  // ------------------------------------------
  // Write data from PLC to RC
  // ------------------------------------------
  30 : IF (( NOT _writeRobotReferenceDynamics.Busy  ) AND 
           ( NOT _writeRobotReferenceDynamics.Error ))
       THEN
         // set command parameter
        _writeRobotReferenceDynamics.ParCmd.DynamicValues :=  ReferenceDynamics;
         // execute command
        _writeRobotReferenceDynamics.Execute := TRUE;
         // set timeout
         SetTimeout(PT := _rTimeout, rTimer := _rTimer);
         // inc step counter
        _rStep := _rStep + 1;
       ELSE
         // check error ? 
         IF (_writeRobotReferenceDynamics.Error)
         THEN
           ErrorID     := _writeRobotReferenceDynamics.ErrorID;
           ErrorAddTxt := _writeRobotReferenceDynamics.ErrorAddTxt;;
         END_IF  
       
         // timeout exceeded ? 
         IF (CheckTimeout(_rTimer) = RobotLibraryConstants.OK)
         THEN
           ErrorID     := RobotLibraryErrorIdEnum.ERR_TIMEOUT_CMD;
           ErrorAddTxt := CONCAT(_stepName, DINT_TO_STRING(_rStep));
         END_IF
       END_IF
 
  31 : IF (( NOT _writeRobotReferenceDynamics.Busy  ) AND
           ( NOT _writeRobotReferenceDynamics.Error ) AND
           (     _writeRobotReferenceDynamics.Done  ))
       THEN
         // execute command
        _writeRobotReferenceDynamics.Execute := FALSE;      
         // update internal ReferenceDynamics data
        _ReferenceDynamics := ReferenceDynamics; 
         // set timeout
         SetTimeout(PT := _rTimeout, rTimer := _rTimer);
         // inc step counter
        _rStep := 10; // -> jump to after startup;           
       ELSE
         // check error ? 
         IF (_writeRobotReferenceDynamics.Error)
         THEN
           SetWarning( WarningID := RobotLibraryWarningIdEnum.WARN_REFERENCE_DYNAMICS_SYNC_FAILED_BY_ERROR_OF_READ_OR_WRITE_CMD, Overwrite := TRUE);    
         END_IF  
       
         // timeout exceeded ? 
         IF (CheckTimeout(_rTimer) = RobotLibraryConstants.OK)
         THEN
           ErrorID     := RobotLibraryErrorIdEnum.ERR_TIMEOUT_CMD;
           ErrorAddTxt := CONCAT(_stepName, DINT_TO_STRING(_rStep));
         END_IF
       END_IF
       
ELSE
  // invalid step
  ErrorID     := RobotLibraryErrorIdEnum.ERR_INVALID_STEP;
  ErrorAddTxt := CONCAT(_stepName , DINT_TO_STRING(_stepCmd));
END_CASE  
                
END_METHOD

METHOD PRIVATE HandleSyncRobotSWLimits
VAR_IN_OUT
   /// Robot assignment of function
  AxesGroup : AxesGroup;
  /// Software limits stored on PLC
  SWLimits  : SWLimits;
END_VAR 

VAR
  /// Internal step counter name
 _stepName        : STRING;    
  /// Internal reference to step counter
 _rStep           : REFERENCE TO DINT;
  /// Internal reference to timer
 _rTimer          : REFERENCE TO TON;
  /// Internal reference to timeout
 _rTimeout        : REFERENCE TO TIME; 
  /// empty data set to reset all DataChanged bits
 _dataChangedNone : AxesGroupStateDataChanged;
END_VAR
                  // Set internal references 
_stepName      :=   '_stepSyncSWLimits = ';
_rStep       REF=    _stepSyncSWLimits;
_rTimer      REF=   _timerSyncSWLimits;
_rTimeout    REF= _timeoutSyncSWLimits;

CASE _rStep
OF    
  0: // Check initialisation configured ?
     IF (( _parCfg.PLC.Parameter.SynchronizationModes.SWLimits[SyncTime.DURING_START_UP] = SyncMode.NO_SYNCHRONIZATION ) AND
         ( _parCfg.PLC.Parameter.SynchronizationModes.SWLimits[SyncTime. AFTER_START_UP] = SyncMode.NO_SYNCHRONIZATION ))
     THEN
       RETURN;
     END_IF

     // Check RC function for sync mode is available ?  
     IF  ((  AxesGroup.State.Initialized                                                  = TRUE                      ) AND  
          (  AxesGroup.State.RobotData.RCSupportedFunctions.WriteRobotSWLimits            = FALSE                     ) AND
         (( _parCfg.PLC.Parameter.SynchronizationModes.SWLimits[SyncTime.DURING_START_UP] = SyncMode.CLIENT_TO_SERVER ) OR
          ( _parCfg.PLC.Parameter.SynchronizationModes.SWLimits[SyncTime. AFTER_START_UP] = SyncMode.CLIENT_TO_SERVER ) OR
          ( _parCfg.PLC.Parameter.SynchronizationModes.SWLimits[SyncTime. AFTER_START_UP] = SyncMode.AUTOMATIC        )))
     THEN
       SetError( ErrorID := RobotLibraryErrorIdEnum.ERR_SYNC_MODE_INVALID, Overwrite := FALSE);
       // Create log entry
       CreateLogMessagePara1 ( Timestamp   := SystemTime,
                               MessageType := MessageType.CMD,
                               Severity    := Severity.DEBUG,
                               MessageCode := 0,
                               MessageText := 'HandleSyncRobotSWLimits: SyncMode needs WriteRobotSWLimits function which is not available on RC',
                               Para1       :=  '');
       RETURN;
     END_IF

     // wait for initialisation done
     IF  ((     AxesGroup.State.RobotData.RCSupportedFunctions .ReadRobotSWLimits ) AND //  ReadRobotSwLimits is mandatory
     //   (     AxesGroup.State.RobotData.RCSupportedFunctions.WriteRobotSWLimits ) AND // WriteRobotSwLimits is optional
          (     AxesGroup.State.Initialized                                       ) AND 
          ( NOT Error                                                             ))  
     THEN
       // Create log entry
       CreateLogMessagePara1 ( Timestamp   := SystemTime,
                               MessageType := MessageType.CMD,
                               Severity    := Severity.DEBUG,
                               MessageCode := 0,
                               MessageText := 'SyncSwLimits: Start initial reading of SwLimits from RC',
                               Para1       :=  '');
       
       // set timeout
       SetTimeout(PT := _rTimeout, rTimer := _rTimer);
       // inc step counter
      _rStep := _rStep + 1;
     END_IF     

     
     // Start read SwLimits
  1: IF (( NOT _readRobotSWLimits.Busy  ) AND 
         ( NOT _readRobotSWLimits.Error ) AND
         ( NOT _readRobotSWLimits.Done  ))
     THEN
       // execute command
      _readRobotSWLimits.Execute := TRUE;
       // set timeout
       SetTimeout(PT := _rTimeout, rTimer := _rTimer);
       // inc step counter
      _rStep := _rStep + 1;
     ELSE
       // check error ? 
       IF ( _readRobotSWLimits.Error )
       THEN
         SetWarning ( WarningID := RobotLibraryWarningIdEnum.WARN_SW_LIMITS_SYNC_FAILED_BY_ERROR_OF_READ_OR_WRITE_CMD, Overwrite := FALSE );           
       END_IF  
       
       // timeout exceeded ? 
       IF (CheckTimeout(_rTimer) = RobotLibraryConstants.OK)
       THEN
         ErrorID     := RobotLibraryErrorIdEnum.ERR_TIMEOUT_CMD;
         ErrorAddTxt := CONCAT(_stepName, DINT_TO_STRING(_rStep));
       END_IF
     END_IF
 
     
     // Wait SwLimits read
  2: IF (( NOT _readRobotSWLimits.Busy  ) AND
         ( NOT _readRobotSWLimits.Error ) AND
         (     _readRobotSWLimits.Done  ))
     THEN
       // reset execution
      _readRobotSWLimits.Execute := FALSE;
       // Copy data
      _swLimits := _readRobotSWLimits.OutCmd.LimitValues;
       // Set plc in sync flag
       AxesGroup.State.SyncStatePlc.InSync.SwLimits := TRUE;
       // inc step counter
      _rStep := _rStep + 1;           

       // Check SwLimits data is equal ? 
       IF ( NOT IsSwLimitsEqual( Data1 := _swLimits, Data2 := SwLimits, IgnoreTimestamp := TRUE))
       THEN
         // Reset plc in sync flag
         AxesGroup.State.SyncStatePlc.InSync.SwLimits := FALSE;
         // Set data changed flag
         AxesGroup.State.DataChanged.SwLimits := TRUE;
         // set timeout
         SetTimeout(PT := _rTimeout, rTimer := _rTimer);
        
         // Create log entry
         CreateLogMessagePara1 ( Timestamp   := SystemTime,
                                 MessageType := MessageType.CMD,
                                 Severity    := Severity.DEBUG,
                                 MessageCode := 0,
                                 MessageText := 'SyncSwLimits: Detected a difference in SwLimits between PLC and RC',
                                 Para1       :=  '');
        
        
         // Check synchronisation is enabled ? 
         IF ( NOT  AxesGroup.State.DataEnableSync.EnableSyncSWLimits )
         THEN
           SetInfo( InfoID := RobotLibraryInfoIdEnum.INFO_SYNC_SWLIMIT_DISABLED, Overwrite := FALSE );
				 END_IF
         
         // Check user interaction needed ?  
         IF ( AxesGroup.Parameter.Plc.Parameter.SyncUserInteraction.SWLimits )
         THEN
           SetWarning ( WarningID := RobotLibraryWarningIdEnum.WARN_SW_LIMITS_SYNC_ERROR, Overwrite := FALSE );                    
				 END_IF
			 END_IF             
     ELSE
       // check error ? 
       IF (_readRobotSWLimits.Error)
       THEN
         // Set warning
         SetWarning( WarningID := RobotLibraryWarningIdEnum.WARN_SW_LIMITS_SYNC_FAILED_BY_ERROR_OF_READ_OR_WRITE_CMD, Overwrite := TRUE);                    
       END_IF  
       
       // timeout exceeded ? 
       IF (CheckTimeout(_rTimer) = RobotLibraryConstants.OK)
       THEN
         ErrorID     := RobotLibraryErrorIdEnum.ERR_TIMEOUT_CMD;
         ErrorAddTxt := CONCAT(_stepName, DINT_TO_STRING(_rStep));
       END_IF
     END_IF
     
     
     // Check synchronisation state ? 
  3: IF ((  NOT AxesGroup.State.DataChanged.SwLimits                                                                                    ) OR 
         (      AxesGroup.Parameter.Plc.Parameter.SynchronizationModes.SWLimits[SyncTime.DURING_START_UP] = SyncMode.NO_SYNCHRONIZATION ))
     THEN
       // Update bit for data in sync
       AxesGroup.State.SyncStatePlc.InSync.SwLimits := NOT AxesGroup.State.DataChanged.SwLimits ;
       // set timeout
       SetTimeout(PT := _rTimeout, rTimer := _rTimer);
       // inc step counter
      _rStep := 10; // -> jump to after startup
            
       // Create log entry
       CreateLogMessagePara1 ( Timestamp   := SystemTime,
                               MessageType := MessageType.CMD,
                               Severity    := Severity.DEBUG,
                               MessageCode := 0,
                               MessageText := 'SyncSwLimits: Synchronization Startup Phase done',
                               Para1       :=  '' );      
     ELSE 
       // Check user interaction needed ? 
       IF ( NOT AxesGroup.Parameter.Plc.Parameter.SyncUserInteraction.SWLimits )
       THEN 
         CASE AxesGroup.Parameter.Plc.Parameter.SynchronizationModes.SWLimits[SyncTime.DURING_START_UP] OF

           SyncMode.SERVER_TO_CLIENT : 

             // Overwrite PLC data with RC data
             SwLimits := _swLimits;            
             // Reset data changed flags
             AxesGroup.State.DataChanged.SwLimits := _dataChangedNone.SwLimits;
             // Reset Synchronizing flag
             AxesGroup.State.Synchronizing.SwLimits := FALSE;
             // Set plc in sync flag
             AxesGroup.State.SyncStatePlc.InSync.SwLimits := TRUE;
             // set timeout
             SetTimeout(PT := _rTimeout, rTimer := _rTimer);
             // inc step counter
            _rStep := 10; // -> jump to after startup         

            // Create log entry
            CreateLogMessagePara2 ( Timestamp   := SystemTime,
                                    MessageType := MessageType.CMD,
                                    Severity    := Severity.DEBUG,
                                    MessageCode := 0,
                                    MessageText := 'SyncSwLimits: Synchronization of SwLimits triggered by StartUp-Compare, SyncMode = {1}, SyncTime = {2}, SyncDirection = RC -> PLC',
                                    Para1       :=  SYNC_MODE_TO_STRING(AxesGroup.Parameter.Plc.Parameter.SynchronizationModes.SWLimits[SyncTime.DURING_START_UP]),
                                    Para2       :=  SYNC_TIME_TO_STRING(SyncTime.DURING_START_UP));
            // Create log entry
            CreateLogMessagePara1 ( Timestamp   := SystemTime,
                                    MessageType := MessageType.CMD,
                                    Severity    := Severity.DEBUG,
                                    MessageCode := 0,
                                    MessageText := 'SyncSwLimits: Applied the initial read SwLimits from RC',
                                    Para1       :=  '' );

				   SyncMode.CLIENT_TO_SERVER : ;

             IF ( AxesGroup.State.DataChanged.SwLimits ) 
             THEN
               // Reset plc in sync flag
               AxesGroup.State.SyncStatePlc.InSync.SwLimits := FALSE;
               // Set Synchronizing flag
               AxesGroup.State.Synchronizing.SwLimits := TRUE;
               // set timeout
               SetTimeout(PT := _rTimeout, rTimer := _rTimer);
               // inc step counter
              _rStep := _rStep +1; // -> write PLC data to RC                  
               // Create log entry
               CreateLogMessagePara2 ( Timestamp   := SystemTime,
                                       MessageType := MessageType.CMD,
                                       Severity    := Severity.DEBUG,
                                       MessageCode := 0,
                                       MessageText := 'SyncSwLimits: Synchronization of SwLimits triggered by StartUp-Compare, SyncMode = {1}, SyncTime = {2}, SyncDirection = PLC -> RC',
                                       Para1       :=  SYNC_MODE_TO_STRING(AxesGroup.Parameter.Plc.Parameter.SynchronizationModes.SWLimits[SyncTime.DURING_START_UP]),
                                       Para2       :=  SYNC_TIME_TO_STRING(SyncTime.DURING_START_UP));
             ELSE
               // Reset data changed flags
               AxesGroup.State.DataChanged.SwLimits := _dataChangedNone.SwLimits;
               // Reset Synchronizing flag
               AxesGroup.State.Synchronizing.SwLimits := FALSE;
               // Set plc in sync flag
               AxesGroup.State.SyncStatePlc.InSync.SwLimits := TRUE;
               // set timeout
               SetTimeout(PT := _rTimeout, rTimer := _rTimer);
               // inc step counter
              _rStep := 10; // -> jump to after startup                  
				     END_IF
         ELSE
           // invalid sync mode for startup
           SetError( ErrorID := RobotLibraryErrorIdEnum.ERR_SYNC_MODE_INVALID, Overwrite := TRUE );
 	       END_CASE
       END_IF
     END_IF  

     
     // Start write SwLimits data  
  4: IF (( NOT _writeRobotSWLimits.Busy  ) AND 
         ( NOT _writeRobotSWLimits.Error ))
     THEN
       // set command parameter
      _writeRobotSWLimits.ParCmd.LimitValues :=  SwLimits;
      _writeRobotSWLimits.ParCmd.ResetToFactoryDefaults := FALSE;
       // execute command
      _writeRobotSWLimits.Execute := TRUE;
       // set timeout
       SetTimeout(PT := _rTimeout, rTimer := _rTimer);
       // inc step counter
      _rStep := _rStep + 1;
     ELSE
       // check error ? 
       IF (_writeRobotSWLimits.Error)
       THEN
         ErrorID     := _writeRobotSWLimits.ErrorID;
         ErrorAddTxt := _writeRobotSWLimits.ErrorAddTxt;;
       END_IF  
       
       // timeout exceeded ? 
       IF (CheckTimeout(_rTimer) = RobotLibraryConstants.OK)
       THEN
         ErrorID     := RobotLibraryErrorIdEnum.ERR_TIMEOUT_CMD;
         ErrorAddTxt := CONCAT(_stepName, DINT_TO_STRING(_rStep));
       END_IF
     END_IF
 
     
     // Wait SwLimits data written ?   
  5: IF (( NOT _writeRobotSWLimits.Busy  ) AND
         ( NOT _writeRobotSWLimits.Error ) AND
         (     _writeRobotSWLimits.Done  ))
     THEN
       // execute command
      _writeRobotSWLimits.Execute := FALSE;
       // apply SwLimits data to internal SwLimits data
      _swLimits := SwLimits;
       // reset data changed bit 
       AxesGroup.State.DataChanged.SwLimits := FALSE;
       // set timeout        
       SetTimeout(PT := _rTimeout, rTimer := _rTimer);
       // dec step counter
      _rStep := _rStep - 2; 
     ELSE
       // check error ? 
       IF (_writeRobotSWLimits.Error)
       THEN
         SetWarning( WarningID := RobotLibraryWarningIdEnum.WARN_SW_LIMITS_SYNC_FAILED_BY_ERROR_OF_READ_OR_WRITE_CMD, Overwrite := TRUE);           
       END_IF  
       
       // timeout exceeded ? 
       IF (CheckTimeout(_rTimer) = RobotLibraryConstants.OK)
       THEN
         ErrorID     := RobotLibraryErrorIdEnum.ERR_TIMEOUT_CMD;
         ErrorAddTxt := CONCAT(_stepName, DINT_TO_STRING(_rStep));
       END_IF
     END_IF

     
  // --------------------------------------------
  // SyncMode after startup : 
  // --------------------------------------------
         
  10 : // check synchronisation active ? 
       IF ( AxesGroup.Parameter.Plc.Parameter.SynchronizationModes.SWLimits[SyncTime.AFTER_START_UP] = SyncMode.NO_SYNCHRONIZATION)
       THEN
         RETURN;
       END_IF

       // compare SwLimits data
       AxesGroup.State.DataChanged.SwLimits := NOT IsSwLimitsEqual( Data1 := SwLimits, Data2 := _swLimits, IgnoreTimestamp := FALSE);

       // Check SwLimits data changed ? 
       IF (AxesGroup.State.DataChanged.SwLimits)
       THEN
         // Create log entry
         CreateLogMessagePara1 ( Timestamp   := SystemTime,
                                 MessageType := MessageType.CMD,
                                 Severity    := Severity.DEBUG,
                                 MessageCode := 0,
                                 MessageText := 'SyncSwLimits: Detected a local change of SwLimits on PLC, SyncTime = {1}',
                                 Para1       :=  SYNC_TIME_TO_STRING(SyncTime.AFTER_START_UP));       
       END_IF

       // Update plc in sync flag
       AxesGroup.State.SyncStatePlc.InSync.SwLimits := NOT AxesGroup.State.DataChanged.SwLimits; 


       // Check synchronization is needed ? 
       IF ( NOT AxesGroup.State.SyncStatePlc.InSync.SwLimits ) XOR  
          ( NOT AxesGroup.State.SyncStateRc .InSync.SwLimits )
       THEN
         CASE AxesGroup.Parameter.Plc.Parameter.SynchronizationModes.SWLimits[SyncTime.AFTER_START_UP] 
         OF         
           // NO_SYNCHRONIZATION
           SyncMode.NO_SYNCHRONIZATION : ; // no further action 
           
           // CLIENT_TO_SERVER
           SyncMode.CLIENT_TO_SERVER :
             // set timeout
             SetTimeout(PT := _rTimeout, rTimer := _rTimer);
             // inc step counter
            _rStep := 11;
  
           // SERVER_TO_CLIENT
           SyncMode.SERVER_TO_CLIENT :
             // set timeout
             SetTimeout(PT := _rTimeout, rTimer := _rTimer);
             // inc step counter
            _rStep := 12;
  
           // AUTOMATIC
           SyncMode.AUTOMATIC : 
             // set timeout
             SetTimeout(PT := _rTimeout, rTimer := _rTimer);
             // inc step counter
            _rStep := 13;
         END_CASE
       ELSE
         // datas changeḍ on both sides ? -> Warning 
         IF (( NOT AxesGroup.State.SyncStatePlc.InSync.SwLimits ) AND  
             ( NOT AxesGroup.State.SyncStateRc .InSync.SwLimits ))
         THEN
           SetWarning( WarningID := RobotLibraryWarningIdEnum.WARN_SW_LIMITS_SYNC_BOTH_SIDES_CHANGED, Overwrite := TRUE);
         END_IF
       END_IF


  // ------------------------------------------
  // SyncMode : CLIENT_TO_SERVER 
  // ------------------------------------------  
  11 : // Conflict triggerd by PLC ?  
       IF ( NOT AxesGroup.State.SyncStatePlc.InSync.SwLimits ) 
       THEN
         // set timeout
         SetTimeout(PT := _rTimeout, rTimer := _rTimer);
         // inc step counter
        _rStep := 30; // -> write PLC data to RC                  
         
         // Create log entry
         CreateLogMessagePara2 ( Timestamp   := SystemTime,
                                 MessageType := MessageType.CMD,
                                 Severity    := Severity.DEBUG,
                                 MessageCode := 0,
                                 MessageText := 'SyncSwLimits: Synchronization of SwLimits triggered by PLC, SyncMode = {1}, SyncTime = {2}, SyncDirection = PLC -> RC',
                                 Para1       :=  SYNC_MODE_TO_STRING(AxesGroup.Parameter.Plc.Parameter.SynchronizationModes.SWLimits[SyncTime.AFTER_START_UP]),
                                 Para2       :=  SYNC_TIME_TO_STRING(SyncTime.AFTER_START_UP));
                                 RETURN;
       END_IF
   
       // Conflict triggered by RC ?
       IF ( NOT AxesGroup.State.SyncStateRc.InSync.SwLimits )
       THEN
         // set timeout
         SetTimeout(PT := _rTimeout, rTimer := _rTimer);
         // inc step counter
        _rStep := 30; // -> write PLC data to RC

         // Create log entry
         CreateLogMessagePara2 ( Timestamp   := SystemTime,
                                 MessageType := MessageType.CMD,
                                 Severity    := Severity.DEBUG,
                                 MessageCode := 0,
                                 MessageText := 'SyncSwLimits: Synchronization of SwLimits triggered by RC, SyncMode = {1}, SyncTime = {2}, SyncDirection = PLC -> RC',
                                 Para1       :=  SYNC_MODE_TO_STRING(AxesGroup.Parameter.Plc.Parameter.SynchronizationModes.SWLimits[SyncTime.AFTER_START_UP]),
                                 Para2       :=  SYNC_TIME_TO_STRING(SyncTime.AFTER_START_UP));
                                 RETURN;
			 END_IF
       
       // set timeout
       SetTimeout(PT := _rTimeout, rTimer := _rTimer);
       // jump back
      _rStep := 10;

       
  // ------------------------------------------
  // SyncMode : SERVER_TO_CLIENT 
  // ------------------------------------------
  12 : // Conflict triggerd by PLC ?  
       IF ( NOT AxesGroup.State.SyncStatePlc.InSync.SwLimits )
       THEN
         // set timeout
         SetTimeout(PT := _rTimeout, rTimer := _rTimer);
         // inc step counter
        _rStep := 20; // -> read RC data and write it to PLC                  

         // Create log entry
         CreateLogMessagePara2 ( Timestamp   := SystemTime,
                                 MessageType := MessageType.CMD,
                                 Severity    := Severity.DEBUG,
                                 MessageCode := 0,
                                 MessageText := 'SyncSwLimits: Synchronization of SwLimits triggered by PLC, SyncMode = {1}, SyncTime = {2}, SyncDirection = RC -> PLC',
                                 Para1       :=  SYNC_MODE_TO_STRING(AxesGroup.Parameter.Plc.Parameter.SynchronizationModes.SWLimits[SyncTime.AFTER_START_UP]),
                                 Para2       :=  SYNC_TIME_TO_STRING(SyncTime.AFTER_START_UP));
                                 RETURN;
       END_IF
   
       // Conflict triggered by RC ?
       IF ( NOT AxesGroup.State.SyncStateRc.InSync.SwLimits )
       THEN
         // set timeout
         SetTimeout(PT := _rTimeout, rTimer := _rTimer);
         // inc step counter
        _rStep := 20; // -> read RC data and write it to PLC

         // Create log entry
         CreateLogMessagePara2 ( Timestamp   := SystemTime,
                                 MessageType := MessageType.CMD,
                                 Severity    := Severity.DEBUG,
                                 MessageCode := 0,
                                 MessageText := 'SyncSwLimits: Synchronization of SwLimits triggered by RC, SyncMode = {1}, SyncTime = {2}, SyncDirection = RC -> PLC',
                                 Para1       :=  SYNC_MODE_TO_STRING(AxesGroup.Parameter.Plc.Parameter.SynchronizationModes.SWLimits[SyncTime.AFTER_START_UP]),
                                 Para2       :=  SYNC_TIME_TO_STRING(SyncTime.AFTER_START_UP));
                                 RETURN;
			 END_IF
       
       // set timeout
       SetTimeout(PT := _rTimeout, rTimer := _rTimer);
       // jump back
      _rStep := 10;
  

  // ------------------------------------------
  // SyncMode : AUTOMATIC 
  // ------------------------------------------
  13 : // Conflict triggerd by PLC ?  
       IF ( NOT AxesGroup.State.SyncStatePlc.InSync.SwLimits )
       THEN
         // set timeout
         SetTimeout(PT := _rTimeout, rTimer := _rTimer);
         // inc step counter
        _rStep := 30; // -> write PLC data to RC                  
         
         // Create log entry
         CreateLogMessagePara2 ( Timestamp   := SystemTime,
                                 MessageType := MessageType.CMD,
                                 Severity    := Severity.DEBUG,
                                 MessageCode := 0,
                                 MessageText := 'SyncSwLimits: Synchronization of SwLimits triggered by PLC, SyncMode = {1}, SyncTime = {2}, SyncDirection = PLC -> RC',
                                 Para1       :=  SYNC_MODE_TO_STRING(AxesGroup.Parameter.Plc.Parameter.SynchronizationModes.SWLimits[SyncTime.AFTER_START_UP]),
                                 Para2       :=  SYNC_TIME_TO_STRING(SyncTime.AFTER_START_UP));
                                 RETURN;
       END_IF
   
       // Conflict triggered by RC ?
       IF ( NOT AxesGroup.State.SyncStateRc.InSync.SwLimits )
       THEN
         // set timeout
         SetTimeout(PT := _rTimeout, rTimer := _rTimer);
         // inc step counter
        _rStep := 20; // -> read RC data an write it to PLC

         // Create log entry
         CreateLogMessagePara2 ( Timestamp   := SystemTime,
                                 MessageType := MessageType.CMD,
                                 Severity    := Severity.DEBUG,
                                 MessageCode := 0,
                                 MessageText := 'SyncSwLimits: Synchronization of SwLimits triggered by RC, SyncMode = {1}, SyncTime = {2}, SyncDirection = RC -> PLC',
                                 Para1       :=  SYNC_MODE_TO_STRING(AxesGroup.Parameter.Plc.Parameter.SynchronizationModes.SWLimits[SyncTime.AFTER_START_UP]),
                                 Para2       :=  SYNC_TIME_TO_STRING(SyncTime.AFTER_START_UP));
                                 RETURN;
			 END_IF
       
       // set timeout
       SetTimeout(PT := _rTimeout, rTimer := _rTimer);
       // jump back
      //_rStep := 10;


  // ------------------------------------------
  // Read Data from RC and write it to PLC
  // ------------------------------------------
  20 : IF (( NOT _readRobotSWLimits.Busy  ) AND 
           ( NOT _readRobotSWLimits.Error ))
       THEN
         // execute command
        _readRobotSWLimits.Execute := TRUE;
         // set timeout
         SetTimeout(PT := _rTimeout, rTimer := _rTimer);
         // inc step counter
        _rStep := _rStep + 1;
       ELSE
         // check error ? 
         IF (_readRobotSWLimits.Error)
         THEN
           ErrorID     := _readRobotSWLimits.ErrorID;
           ErrorAddTxt := _readRobotSWLimits.ErrorAddTxt;
         END_IF  
       
         // timeout exceeded ? 
         IF (CheckTimeout(_rTimer) = RobotLibraryConstants.OK)
         THEN
           ErrorID     := RobotLibraryErrorIdEnum.ERR_TIMEOUT_CMD;
           ErrorAddTxt := CONCAT(_stepName, DINT_TO_STRING(_rStep));
         END_IF
       END_IF
 
  21 : IF (( NOT _readRobotSWLimits.Busy  ) AND
           ( NOT _readRobotSWLimits.Error ) AND
           (     _readRobotSWLimits.Done  ))
       THEN
         // reset execution
        _readRobotSWLimits.Execute := FALSE;
         // update internal SwLimits data
         SwLimits := _readRobotSWLimits.OutCmd.LimitValues;         
        _swLimits := _readRobotSWLimits.OutCmd.LimitValues;
         // set timeout
         SetTimeout(PT := _rTimeout, rTimer := _rTimer);
         // inc step counter
        _rStep := 10; // -> jump to after startup           
       ELSE
         // check error ? 
         IF (_readRobotSWLimits.Error)
         THEN
           ErrorID     := _readRobotSWLimits.ErrorID;
           ErrorAddTxt := _readRobotSWLimits.ErrorAddTxt;           
         END_IF  
       
         // timeout exceeded ? 
         IF (CheckTimeout(_rTimer) = RobotLibraryConstants.OK)
         THEN
           ErrorID     := RobotLibraryErrorIdEnum.ERR_TIMEOUT_CMD;
           ErrorAddTxt := CONCAT(_stepName, DINT_TO_STRING(_rStep));
         END_IF
       END_IF


  // ------------------------------------------
  // Write data from PLC to RC
  // ------------------------------------------
  30 : IF (( NOT _writeRobotSWLimits.Busy  ) AND 
           ( NOT _writeRobotSWLimits.Error ))
       THEN
         // set command parameter
        _writeRobotSWLimits.ParCmd.ResetToFactoryDefaults := FALSE;      
        _writeRobotSWLimits.ParCmd.LimitValues :=  SwLimits;
         // execute command
        _writeRobotSWLimits.Execute := TRUE;
         // set timeout
         SetTimeout(PT := _rTimeout, rTimer := _rTimer);
         // inc step counter
        _rStep := _rStep + 1;
       ELSE
         // check error ? 
         IF (_writeRobotSWLimits.Error)
         THEN
           ErrorID     := _writeRobotSWLimits.ErrorID;
           ErrorAddTxt := _writeRobotSWLimits.ErrorAddTxt;;
         END_IF  
       
         // timeout exceeded ? 
         IF (CheckTimeout(_rTimer) = RobotLibraryConstants.OK)
         THEN
           ErrorID     := RobotLibraryErrorIdEnum.ERR_TIMEOUT_CMD;
           ErrorAddTxt := CONCAT(_stepName, DINT_TO_STRING(_rStep));
         END_IF
       END_IF
 
  31 : IF (( NOT _writeRobotSWLimits.Busy  ) AND
           ( NOT _writeRobotSWLimits.Error ) AND
           (     _writeRobotSWLimits.Done  ))
       THEN
         // execute command
        _writeRobotSWLimits.Execute := FALSE;      
         // update internal SwLimits data
        _swLimits := SwLimits; 
         // set timeout
         SetTimeout(PT := _rTimeout, rTimer := _rTimer);
         // inc step counter
        _rStep := 10; // -> jump to after startup;           
       ELSE
         // check error ? 
         IF (_writeRobotSWLimits.Error)
         THEN
           SetWarning( WarningID := RobotLibraryWarningIdEnum.WARN_SW_LIMITS_SYNC_FAILED_BY_ERROR_OF_READ_OR_WRITE_CMD, Overwrite := TRUE);    
         END_IF  
       
         // timeout exceeded ? 
         IF (CheckTimeout(_rTimer) = RobotLibraryConstants.OK)
         THEN
           ErrorID     := RobotLibraryErrorIdEnum.ERR_TIMEOUT_CMD;
           ErrorAddTxt := CONCAT(_stepName, DINT_TO_STRING(_rStep));
         END_IF
       END_IF
       
ELSE
  // invalid step
  ErrorID     := RobotLibraryErrorIdEnum.ERR_INVALID_STEP;
  ErrorAddTxt := CONCAT(_stepName , DINT_TO_STRING(_stepCmd));
END_CASE  
                
END_METHOD

METHOD PRIVATE HandleSyncToolData
VAR_IN_OUT
   /// Robot assignment of function
  AxesGroup : AxesGroup;
  /// ToolData stored on PLC.For more information refer to 5.5.6.4
  ToolData  : ARRAY[*] OF Tool;
END_VAR 

VAR
  /// Internal step counter name
 _stepName        : STRING;    
  /// Internal reference to step counter
 _rStep           : REFERENCE TO DINT;
  /// Internal reference to timer
 _rTimer          : REFERENCE TO TON;
  /// Internal reference to timeout
 _rTimeout        : REFERENCE TO TIME; 
  /// Internal reference to synchroniztion index
 _rSyncIdx        : REFERENCE TO USINT;
  /// internal bit for condition found
 _found           : BOOL;
  /// empty data set to reset all DataChanged bits
 _dataChangedNone : AxesGroupStateDataChanged; 
  /// internal index for loops
 _idx             : DINT;
END_VAR
                  // Set internal references 
_stepName      :=   '_stepSyncToolData = ';
_rStep       REF=    _stepSyncToolData;
_rTimer      REF=   _timerSyncToolData;
_rTimeout    REF= _timeoutSyncToolData;
_rSyncIdx    REF=     _syncIdxToolData;


CASE _rStep
OF    
  0: // Check initialisation configured ?
     IF (( _parCfg.PLC.Parameter.SynchronizationModes.Tool[SyncTime.DURING_START_UP] = SyncMode.NO_SYNCHRONIZATION ) AND
         ( _parCfg.PLC.Parameter.SynchronizationModes.Tool[SyncTime. AFTER_START_UP] = SyncMode.NO_SYNCHRONIZATION ))
     THEN
       RETURN;
     END_IF
     
     // Check More Data on RC than on PLC -> Synchronization not possible
     IF (AxesGroup.State.ConfigurationData.HighestToolIndex > AxesGroup.SystemData.ToolDataCount)
     THEN
       SetError( ErrorID := RobotLibraryErrorIdEnum.ERR_SYNC_TOOL_COUNT_RC_HIGHER_THAN_PLC, Overwrite := FALSE);
       RETURN;
		 END_IF

     // wait for initialisation done
     IF  ((     AxesGroup.State.RobotData.RCSupportedFunctions. ReadToolData ) AND
          (     AxesGroup.State.RobotData.RCSupportedFunctions.WriteToolData ) AND
          (     AxesGroup.State.Initialized                                  ) AND 
          ( NOT Error                                                        ))  
     THEN
       // Check PLC tools < RC tools and SyncTool enabled ?    
       IF (( AxesGroup.State.DataEnableSync.EnableSyncTool      = TRUE                             )  AND
           ( AxesGroup.Parameter.Rob.Parameter.HighestToolIndex > AxesGroup.SystemData.ToolDataMax ))        
       THEN
         SetWarning( WarningID := RobotLibraryWarningIdEnum.WARN_TOOL_DATA_ARRAY_TOO_SHORT, Overwrite := TRUE);
       END_IF

       // Create log entry
       CreateLogMessagePara1 ( Timestamp   := SystemTime,
                               MessageType := MessageType.CMD,
                               Severity    := Severity.DEBUG,
                               MessageCode := 0,
                               MessageText := 'SyncToolData: Start initial reading of ToolData from RC',
                               Para1       :=  '');
       
       // init tool number
      _rSyncIdx := DINT_TO_USINT(AxesGroup.SystemData.ToolDataMin); 
       // init count of unsynchronized elements
       AxesGroup.State.SyncStatePlc.UnSyncNo.Tool := 0;
       // set timeout
       SetTimeout(PT := _rTimeout, rTimer := _rTimer);
       // inc step counter
      _rStep := _rStep + 1;
     END_IF     

     
     // Start read ToolData
  1: IF (( NOT _readToolData.Busy  ) AND 
         ( NOT _readToolData.Error ) AND
         ( NOT _readToolData.Done  ))
     THEN
       // set command parameter
      _readToolData.ParCmd.ToolNo := _rSyncIdx;      
       // execute command
      _readToolData.Execute := TRUE;
       // set timeout
       SetTimeout(PT := _rTimeout, rTimer := _rTimer);
       // inc step counter
      _rStep := _rStep + 1;
     ELSE
       // check error ? 
       IF ( _readToolData.Error ) AND ( WarningID = RobotLibraryWarningIdEnum.NO_WARNING )
       THEN
         SetWarning( WarningID := RobotLibraryWarningIdEnum.WARN_TOOL_SYNC_FAILED_BY_ERROR_OF_READ_OR_WRITE_CMD, Overwrite := TRUE);           
       END_IF  
       
       // timeout exceeded ? 
       IF (CheckTimeout(_rTimer) = RobotLibraryConstants.OK)
       THEN
         ErrorID     := RobotLibraryErrorIdEnum.ERR_TIMEOUT_CMD;
         ErrorAddTxt := CONCAT(_stepName, DINT_TO_STRING(_rStep));
       END_IF
     END_IF
 
     
     // Wait Tooldata read
  2: IF (( NOT _readToolData.Busy  ) AND
         ( NOT _readToolData.Error ) AND
         (     _readToolData.Done  ))
     THEN
       // reset execution
      _readToolData.Execute := FALSE;
       // set available bit
      _toolData[_rSyncIdx].Available := TRUE; 
       ToolData[_rSyncIdx].Available := TRUE;      
       // Copy data
      _toolData[_rSyncIdx].Data := _readToolData.OutCmd.ToolData;

       // Check tool data is equal ? 
       IF ( NOT IsToolDataEqual( Data1 := _toolData[_rSyncIdx].Data, Data2 := ToolData[_rSyncIdx].Data, IgnoreTimestamp := TRUE))
       THEN
         // Reset plc in sync flag
         AxesGroup.State.SyncStatePlc.InSync.Tool := FALSE;
         // Set data changed flag
         AxesGroup.State.DataChanged.Tool[_rSyncIdx] := TRUE;
         // inc count of unsynchronised plc tools
         AxesGroup.State.SyncStatePlc.UnSyncNo.Tool := AxesGroup.State.SyncStatePlc.UnSyncNo.Tool + 1;
        
         // Create log entry
         CreateLogMessagePara1 ( Timestamp   := SystemTime,
                                 MessageType := MessageType.CMD,
                                 Severity    := Severity.DEBUG,
                                 MessageCode := 0,
                                 MessageText := 'SyncToolData: Detected a difference in Tool[{1}] between PLC and RC',
                                 Para1       :=  DINT_TO_STRING(_rSyncIdx));
        
        
         // Check synchronisation is enabled ? 
         IF ( NOT AxesGroup.State.DataEnableSync.EnableSyncTool ) AND (InfoID = RobotLibraryInfoIdEnum.NO_INFO )
         THEN
           SetInfo( InfoID := RobotLibraryInfoIdEnum.INFO_SYNC_TOOL_DATA_DISABLED, Overwrite := TRUE);
				 END_IF
         
         // Check user interaction needed ?  
         IF ( AxesGroup.Parameter.PLC.Parameter.SyncUserInteraction.Tool ) AND ( WarningID = RobotLibraryWarningIdEnum.NO_WARNING )
         THEN
           SetWarning( WarningID := RobotLibraryWarningIdEnum.WARN_TOOL_NUMBER_SYNC_ERROR, Overwrite :=  TRUE);                    
				 END_IF
			 END_IF
             
       // Check all tools read ? 
       IF ( _rSyncIdx < AxesGroup.State.UnifiedToolIndex )
       THEN
         // set timeout
         SetTimeout(PT := _rTimeout, rTimer := _rTimer);
         // inc tool index
        _rSyncIdx := _rSyncIdx + 1;
         // dec step counter
        _rStep := _rStep - 1;
       ELSE
         // set timeout
         SetTimeout(PT := _rTimeout, rTimer := _rTimer);
         // inc step counter
        _rStep := _rStep + 1;           
       END_IF
     ELSE
       // check error ? 
       IF (_readToolData.Error)
       THEN
         // Set warning
         SetWarning( WarningID := RobotLibraryWarningIdEnum.WARN_TOOL_SYNC_FAILED_BY_ERROR_OF_READ_OR_WRITE_CMD, Overwrite := TRUE);                    
         // reset available bit
         ToolData[_rSyncIdx].Available := FALSE;
        _toolData[_rSyncIdx].Available := FALSE;
       END_IF  
       
       // timeout exceeded ? 
       IF (CheckTimeout(_rTimer) = RobotLibraryConstants.OK)
       THEN
         ErrorID     := RobotLibraryErrorIdEnum.ERR_TIMEOUT_CMD;
         ErrorAddTxt := CONCAT(_stepName, DINT_TO_STRING(_rStep));
       END_IF
     END_IF
     
     
     // Check synchronisation state ? 
  3: IF (( AxesGroup.State.SyncStatePlc.UnSyncNo.Tool                                            = 0                           ) OR 
         ( AxesGroup.Parameter.Plc.Parameter.SynchronizationModes.Tool[SyncTime.DURING_START_UP] = SyncMode.NO_SYNCHRONIZATION ))
     THEN
       // Update bit for data in sync
       AxesGroup.State.SyncStatePlc.InSync.Tool := (AxesGroup.State.SyncStatePlc.UnSyncNo.Tool = 0);
       // set timeout
       SetTimeout(PT := _rTimeout, rTimer := _rTimer);
       // inc step counter
      _rStep := 10; // -> jump to after startup
            
       // Create log entry
       CreateLogMessagePara1 ( Timestamp   := SystemTime,
                               MessageType := MessageType.CMD,
                               Severity    := Severity.DEBUG,
                               MessageCode := 0,
                               MessageText := 'SyncToolData: Synchronization Startup Phase done',
                               Para1       :=  '' );      
     ELSE 
       // Check user interaction needed ? 
       IF ( NOT AxesGroup.Parameter.PLC.Parameter.SyncUserInteraction.Tool )
       THEN
         CASE AxesGroup.Parameter.Plc.Parameter.SynchronizationModes.Tool[SyncTime.DURING_START_UP] OF

           SyncMode.SERVER_TO_CLIENT : 

           
             FOR _idx := AxesGroup.SystemData.ToolDataMin TO AxesGroup.SystemData.ToolDataMax
             DO
               // Overwrite PLC data with RC data
               ToolData[_idx] := _toolData[_idx];            
						 END_FOR
             // Reset data changed flags
             AxesGroup.State.DataChanged.Tool := _dataChangedNone.Tool;
             // Reset Synchronizing flag
             AxesGroup.State.Synchronizing.Tool := FALSE;
             // Set plc in sync flag
             AxesGroup.State.SyncStatePlc.InSync.Tool := TRUE;
             // Reset count of unsynchronised plc tools
             AxesGroup.State.SyncStatePlc.UnSyncNo.Tool := 0;            
             // set timeout
             SetTimeout(PT := _rTimeout, rTimer := _rTimer);
             // inc step counter
            _rStep := 10; // -> jump to after startup         

            // Create log entry
            CreateLogMessagePara3 ( Timestamp   := SystemTime,
                                    MessageType := MessageType.CMD,
                                    Severity    := Severity.DEBUG,
                                    MessageCode := 0,
                                    MessageText := 'SyncToolData: Synchronization of Tools triggered by StartUp-Compare, SyncMode = {2}, SyncTime = {3}, SyncDirection = RC -> PLC',
                                    Para1       :=  DINT_TO_STRING(_rSyncIdx),
                                    Para2       :=  SYNC_MODE_TO_STRING(AxesGroup.Parameter.Plc.Parameter.SynchronizationModes.Tool[SyncTime.DURING_START_UP]),
                                    Para3       :=  SYNC_TIME_TO_STRING(SyncTime.DURING_START_UP));
            // Create log entry
            CreateLogMessagePara1 ( Timestamp   := SystemTime,
                                    MessageType := MessageType.CMD,
                                    Severity    := Severity.DEBUG,
                                    MessageCode := 0,
                                    MessageText := 'SyncToolData: Applied the initial read tool data from RC',
                                    Para1       :=  '' );

				   SyncMode.CLIENT_TO_SERVER : ;

             // Check conflicts to solve ? 
             FOR _rSyncIdx := 0 TO AxesGroup.State.UnifiedToolIndex
             DO
               IF ( AxesGroup.State.DataChanged.Tool[_rSyncIdx] )
               THEN
                _found := TRUE;
                 EXIT;
		  			   END_IF
             END_FOR
           
             IF ( _found ) 
             THEN
               // Reset plc in sync flag
               AxesGroup.State.SyncStatePlc.InSync.Tool := FALSE;
               // Set Synchronizing flag
               AxesGroup.State.Synchronizing.Tool := TRUE;
               // set timeout
               SetTimeout(PT := _rTimeout, rTimer := _rTimer);
               // inc step counter
              _rStep := _rStep +1; // -> write PLC data to RC                  
               // Create log entry
               CreateLogMessagePara3 ( Timestamp   := SystemTime,
                                       MessageType := MessageType.CMD,
                                       Severity    := Severity.DEBUG,
                                       MessageCode := 0,
                                       MessageText := 'SyncToolData: Synchronization of Tool[{1}] triggered by StartUp-Compare, SyncMode = {2}, SyncTime = {3}, SyncDirection = PLC -> RC',
                                       Para1       :=  DINT_TO_STRING(_rSyncIdx),
                                       Para2       :=  SYNC_MODE_TO_STRING(AxesGroup.Parameter.Plc.Parameter.SynchronizationModes.Tool[SyncTime.DURING_START_UP]),
                                       Para3       :=  SYNC_TIME_TO_STRING(SyncTime.DURING_START_UP));
             ELSE
               // Reset data changed flags
               AxesGroup.State.DataChanged.Tool := _dataChangedNone.Tool;
               // Reset Synchronizing flag
               AxesGroup.State.Synchronizing.Tool := FALSE;
               // Set plc in sync flag
               AxesGroup.State.SyncStatePlc.InSync.Tool := TRUE;
               // Reset count of unsynchronised tools
               AxesGroup.State.SyncStatePlc.UnSyncNo.Tool := 0;
               // set timeout
               SetTimeout(PT := _rTimeout, rTimer := _rTimer);
               // inc step counter
              _rStep := 10; // -> jump to after startup                  
				     END_IF
         ELSE
           // invalid sync mode for startup
           SetError( ErrorID := RobotLibraryErrorIdEnum.ERR_SYNC_MODE_INVALID, Overwrite := TRUE );
 	       END_CASE
       END_IF
     END_IF  

     
     // Start write tool data  
  4: IF (( NOT _writeToolData.Busy  ) AND 
         ( NOT _writeToolData.Error ))
     THEN
       // set command parameter
      _writeToolData.ParCmd.ToolNo   := _rSyncIdx;      
      _writeToolData.ParCmd.ToolData :=  ToolData[_rSyncIdx].Data;
       // execute command
      _writeToolData.Execute := TRUE;
       // set timeout
       SetTimeout(PT := _rTimeout, rTimer := _rTimer);
       // inc step counter
      _rStep := _rStep + 1;
     ELSE
       // check error ? 
       IF (_writeToolData.Error)
       THEN
         ErrorID     := _writeToolData.ErrorID;
         ErrorAddTxt := _writeToolData.ErrorAddTxt;;
       END_IF  
       
       // timeout exceeded ? 
       IF (CheckTimeout(_rTimer) = RobotLibraryConstants.OK)
       THEN
         ErrorID     := RobotLibraryErrorIdEnum.ERR_TIMEOUT_CMD;
         ErrorAddTxt := CONCAT(_stepName, DINT_TO_STRING(_rStep));
       END_IF
     END_IF
 
     
     // Wait tool data written ?   
  5: IF (( NOT _writeToolData.Busy  ) AND
         ( NOT _writeToolData.Error ) AND
         (     _writeToolData.Done  ))
     THEN
       // execute command
      _writeToolData.Execute := FALSE;
       // apply tool data to internal tool data
      _toolData[_rSyncIdx] := ToolData[_rSyncIdx];
       // reset data changed bit 
       AxesGroup.State.DataChanged.Tool[_rSyncIdx] := FALSE;
       // dec count of unsynchronised tools
       AxesGroup.State.SyncStatePlc.UnSyncNo.Tool := AxesGroup.State.SyncStatePlc.UnSyncNo.Tool - 1;
       // set timeout        
       SetTimeout(PT := _rTimeout, rTimer := _rTimer);
       // dec step counter
      _rStep := _rStep - 2; 
     ELSE
       // check error ? 
       IF (_writeToolData.Error)
       THEN
         SetWarning( WarningID := RobotLibraryWarningIdEnum.WARN_TOOL_SYNC_FAILED_BY_ERROR_OF_READ_OR_WRITE_CMD, Overwrite := TRUE);           
       END_IF  
       
       // timeout exceeded ? 
       IF (CheckTimeout(_rTimer) = RobotLibraryConstants.OK)
       THEN
         ErrorID     := RobotLibraryErrorIdEnum.ERR_TIMEOUT_CMD;
         ErrorAddTxt := CONCAT(_stepName, DINT_TO_STRING(_rStep));
       END_IF
     END_IF

     
  // --------------------------------------------
  // SyncMode after startup : 
  // --------------------------------------------
         
  10 :// check synchronisation active ? 
       IF ( AxesGroup.Parameter.Plc.Parameter.SynchronizationModes.Tool[SyncTime.AFTER_START_UP] = SyncMode.NO_SYNCHRONIZATION)
       THEN
         RETURN;
       END_IF

       // reset count of unsynchronised tools
       AxesGroup.State.SyncStatePlc.UnSyncNo.Tool := 0;

       // Check all tool datas
       FOR _rSyncIdx := 0 TO AxesGroup.State.UnifiedToolIndex
       DO
         // compare tool data
         AxesGroup.State.DataChanged.Tool[_rSyncIdx] := NOT IsToolDataEqual( Data1 := ToolData[_rSyncIdx].Data, Data2 := _toolData[_rSyncIdx].Data, IgnoreTimestamp := FALSE);

         // Check Tool data changed ? 
         IF (AxesGroup.State.DataChanged.Tool[_rSyncIdx])
         THEN
           // inc count of unsynchronised plc tools
           AxesGroup.State.SyncStatePlc.UnSyncNo.Tool := AxesGroup.State.SyncStatePlc.UnSyncNo.Tool + 1;
           // Create log entry
           CreateLogMessagePara2 ( Timestamp   := SystemTime,
                                   MessageType := MessageType.CMD,
                                   Severity    := Severity.DEBUG,
                                   MessageCode := 0,
                                   MessageText := 'SyncToolData: Detected a local change of Tool[{1}] on PLC, SyncTime = {2}',
                                   Para1       :=  DINT_TO_STRING(_rSyncIdx),    
                                   Para2       :=  SYNC_TIME_TO_STRING(SyncTime.AFTER_START_UP));       
				 END_IF

         // Update plc in sync flag
         AxesGroup.State.SyncStatePlc.InSync.Tool := (AxesGroup.State.SyncStatePlc.UnSyncNo.Tool = 0); 
	     END_FOR

       // Check synchronization is needed ? 
       IF ( NOT AxesGroup.State.SyncStatePlc.InSync.Tool ) XOR  
          ( NOT AxesGroup.State.SyncStateRc .InSync.Tool )
       THEN
         CASE AxesGroup.Parameter.Plc.Parameter.SynchronizationModes.Tool[SyncTime.AFTER_START_UP] 
         OF         
           // NO_SYNCHRONIZATION
           SyncMode.NO_SYNCHRONIZATION : ; // no further action 
           
           // CLIENT_TO_SERVER
           SyncMode.CLIENT_TO_SERVER :
             // set timeout
             SetTimeout(PT := _rTimeout, rTimer := _rTimer);
             // inc step counter
            _rStep := 11;
  
           // SERVER_TO_CLIENT
           SyncMode.SERVER_TO_CLIENT :
             // set timeout
             SetTimeout(PT := _rTimeout, rTimer := _rTimer);
             // inc step counter
            _rStep := 12;
  
           // AUTOMATIC
           SyncMode.AUTOMATIC : 
             // set timeout
             SetTimeout(PT := _rTimeout, rTimer := _rTimer);
             // inc step counter
            _rStep := 13;
         END_CASE
       ELSE
         // datas changeḍ on both sides ? -> Warning 
         IF (( NOT AxesGroup.State.SyncStatePlc.InSync.Tool ) AND  
             ( NOT AxesGroup.State.SyncStateRc .InSync.Tool ))
         THEN
           SetWarning( WarningID := RobotLibraryWarningIdEnum.WARN_TOOL_SYNC_BOTH_SIDES_CHANGED, Overwrite := TRUE);
         END_IF
       END_IF


  // ------------------------------------------
  // SyncMode : CLIENT_TO_SERVER 
  // ------------------------------------------  
  11 : // Conflict triggerd by PLC ?  
       IF ( NOT AxesGroup.State.SyncStatePlc.InSync.Tool )
       THEN
         // search for changed index  
         FOR _rSyncIdx := 0 TO AxesGroup.State.UnifiedToolIndex
         DO
           IF ( AxesGroup.State.DataChanged.Tool[_rSyncIdx] )
           THEN
             // set timeout
             SetTimeout(PT := _rTimeout, rTimer := _rTimer);
             // inc step counter
            _rStep := 30; // -> write PLC data to RC                  
             EXIT;             
					 END_IF
         END_FOR
         
         // Create log entry
         CreateLogMessagePara3 ( Timestamp   := SystemTime,
                                 MessageType := MessageType.CMD,
                                 Severity    := Severity.DEBUG,
                                 MessageCode := 0,
                                 MessageText := 'SyncToolData: Synchronization of Tool[{1}] triggered by PLC, SyncMode = {2}, SyncTime = {3}, SyncDirection = PLC -> RC',
                                 Para1       :=  DINT_TO_STRING(_rSyncIdx),
                                 Para2       :=  SYNC_MODE_TO_STRING(AxesGroup.Parameter.Plc.Parameter.SynchronizationModes.Tool[SyncTime.AFTER_START_UP]),
                                 Para3       :=  SYNC_TIME_TO_STRING(SyncTime.AFTER_START_UP));
                                 RETURN;
       END_IF
   
       // Conflict triggered by RC ?
       IF ( NOT AxesGroup.State.SyncStateRc.InSync.Tool )
       THEN
         // get changed index 
        _rSyncIdx :=  LIMIT(0, AxesGroup.State.SyncStateRc.UnSyncNo.Tool, AxesGroup.State.UnifiedToolIndex);
         // set timeout
         SetTimeout(PT := _rTimeout, rTimer := _rTimer);
         // inc step counter
        _rStep := 30; // -> write PLC data to RC

         // Create log entry
         CreateLogMessagePara3 ( Timestamp   := SystemTime,
                                 MessageType := MessageType.CMD,
                                 Severity    := Severity.DEBUG,
                                 MessageCode := 0,
                                 MessageText := 'SyncToolData: Synchronization of Tool[{1}] triggered by RC, SyncMode = {2}, SyncTime = {3}, SyncDirection = PLC -> RC',
                                 Para1       :=  DINT_TO_STRING(_rSyncIdx),
                                 Para2       :=  SYNC_MODE_TO_STRING(AxesGroup.Parameter.Plc.Parameter.SynchronizationModes.Tool[SyncTime.AFTER_START_UP]),
                                 Para3       :=  SYNC_TIME_TO_STRING(SyncTime.AFTER_START_UP));
                                 RETURN;
			 END_IF
       
       // set timeout
       SetTimeout(PT := _rTimeout, rTimer := _rTimer);
       // jump back
      _rStep := 10;

       
  // ------------------------------------------
  // SyncMode : SERVER_TO_CLIENT 
  // ------------------------------------------
  12 : // Conflict triggerd by PLC ?  
       IF ( NOT AxesGroup.State.SyncStatePlc.InSync.Tool )
       THEN
         // search for changed index  
         FOR _rSyncIdx := 0 TO AxesGroup.State.UnifiedToolIndex
         DO
           IF ( AxesGroup.State.DataChanged.Tool[_rSyncIdx] )
           THEN
             // set timeout
             SetTimeout(PT := _rTimeout, rTimer := _rTimer);
             // inc step counter
            _rStep := 20; // -> read RC data and write it to PLC                  
             EXIT;
					 END_IF
         END_FOR

         // Create log entry
         CreateLogMessagePara3 ( Timestamp   := SystemTime,
                                 MessageType := MessageType.CMD,
                                 Severity    := Severity.DEBUG,
                                 MessageCode := 0,
                                 MessageText := 'SyncToolData: Synchronization of Tool[{1}] triggered by PLC, SyncMode = {2}, SyncTime = {3}, SyncDirection = RC -> PLC',
                                 Para1       :=  DINT_TO_STRING(_rSyncIdx),
                                 Para2       :=  SYNC_MODE_TO_STRING(AxesGroup.Parameter.Plc.Parameter.SynchronizationModes.Tool[SyncTime.AFTER_START_UP]),
                                 Para3       :=  SYNC_TIME_TO_STRING(SyncTime.AFTER_START_UP));
                                 RETURN;
       END_IF
   
       // Conflict triggered by RC ?
       IF ( NOT AxesGroup.State.SyncStateRc.InSync.Tool )
       THEN
         // get changed index 
        _rSyncIdx := LIMIT(0, AxesGroup.State.SyncStateRc.UnSyncNo.Tool, AxesGroup.State.UnifiedToolIndex);
         // set timeout
         SetTimeout(PT := _rTimeout, rTimer := _rTimer);
         // inc step counter
        _rStep := 20; // -> read RC data and write it to PLC

         // Create log entry
         CreateLogMessagePara3 ( Timestamp   := SystemTime,
                                 MessageType := MessageType.CMD,
                                 Severity    := Severity.DEBUG,
                                 MessageCode := 0,
                                 MessageText := 'SyncToolData: Synchronization of Tool[{1}] triggered by RC, SyncMode = {2}, SyncTime = {3}, SyncDirection = RC -> PLC',
                                 Para1       :=  DINT_TO_STRING(_rSyncIdx),
                                 Para2       :=  SYNC_MODE_TO_STRING(AxesGroup.Parameter.Plc.Parameter.SynchronizationModes.Tool[SyncTime.AFTER_START_UP]),
                                 Para3       :=  SYNC_TIME_TO_STRING(SyncTime.AFTER_START_UP));
                                 RETURN;
			 END_IF
       
       // set timeout
       SetTimeout(PT := _rTimeout, rTimer := _rTimer);
       // jump back
      _rStep := 10;
  

  // ------------------------------------------
  // SyncMode : AUTOMATIC 
  // ------------------------------------------
  13 : // Conflict triggerd by PLC ?  
       IF ( NOT AxesGroup.State.SyncStatePlc.InSync.Tool )
       THEN
         // search for changed index  
         FOR _rSyncIdx := 0 TO AxesGroup.State.UnifiedToolIndex
         DO
           IF ( AxesGroup.State.DataChanged.Tool[_rSyncIdx] )
           THEN
             // set timeout
             SetTimeout(PT := _rTimeout, rTimer := _rTimer);
             // inc step counter
            _rStep := 30; // -> write PLC data to RC                  
             EXIT;
					 END_IF
         END_FOR
         
         // Create log entry
         CreateLogMessagePara3 ( Timestamp   := SystemTime,
                                 MessageType := MessageType.CMD,
                                 Severity    := Severity.DEBUG,
                                 MessageCode := 0,
                                 MessageText := 'SyncToolData: Synchronization of Tool[{1}] triggered by PLC, SyncMode = {2}, SyncTime = {3}, SyncDirection = PLC -> RC',
                                 Para1       :=  DINT_TO_STRING(_rSyncIdx),
                                 Para2       :=  SYNC_MODE_TO_STRING(AxesGroup.Parameter.Plc.Parameter.SynchronizationModes.Tool[SyncTime.AFTER_START_UP]),
                                 Para3       :=  SYNC_TIME_TO_STRING(SyncTime.AFTER_START_UP));
                                 RETURN;
       END_IF
   
       // Conflict triggered by RC ?
       IF ( NOT AxesGroup.State.SyncStateRc.InSync.Tool )
       THEN
         // get changed index 
        _rSyncIdx := LIMIT(0, AxesGroup.State.SyncStateRc.UnSyncNo.Tool, AxesGroup.State.UnifiedToolIndex);
         // set timeout
         SetTimeout(PT := _rTimeout, rTimer := _rTimer);
         // inc step counter
        _rStep := 20; // -> read RC data an write it to PLC

         // Create log entry
         CreateLogMessagePara3 ( Timestamp   := SystemTime,
                                 MessageType := MessageType.CMD,
                                 Severity    := Severity.DEBUG,
                                 MessageCode := 0,
                                 MessageText := 'SyncToolData: Synchronization of Tool[{1}] triggered by RC, SyncMode = {2}, SyncTime = {3}, SyncDirection = RC -> PLC',
                                 Para1       :=  DINT_TO_STRING(_rSyncIdx),
                                 Para2       :=  SYNC_MODE_TO_STRING(AxesGroup.Parameter.Plc.Parameter.SynchronizationModes.Tool[SyncTime.AFTER_START_UP]),
                                 Para3       :=  SYNC_TIME_TO_STRING(SyncTime.AFTER_START_UP));
                                 RETURN;
			 END_IF
       
       // set timeout
       SetTimeout(PT := _rTimeout, rTimer := _rTimer);
       // jump back
      //_rStep := 10;


  // ------------------------------------------
  // Read Data from RC and write it to PLC
  // ------------------------------------------
  20 : IF (( NOT _readToolData.Busy  ) AND 
           ( NOT _readToolData.Error ))
       THEN
         // set command parameter
        _readToolData.ParCmd.ToolNo := _rSyncIdx;      
         // execute command
        _readToolData.Execute := TRUE;
         // set timeout
         SetTimeout(PT := _rTimeout, rTimer := _rTimer);
         // inc step counter
        _rStep := _rStep + 1;
       ELSE
         // check error ? 
         IF (_readToolData.Error)
         THEN
           ErrorID     := _readToolData.ErrorID;
           ErrorAddTxt := _readToolData.ErrorAddTxt;
         END_IF  
       
         // timeout exceeded ? 
         IF (CheckTimeout(_rTimer) = RobotLibraryConstants.OK)
         THEN
           ErrorID     := RobotLibraryErrorIdEnum.ERR_TIMEOUT_CMD;
           ErrorAddTxt := CONCAT(_stepName, DINT_TO_STRING(_rStep));
         END_IF
       END_IF
 
  21 : IF (( NOT _readToolData.Busy  ) AND
           ( NOT _readToolData.Error ) AND
           (     _readToolData.Done  ))
       THEN
         // reset execution
        _readToolData.Execute := FALSE;
         // update internal tool data
         ToolData[_rSyncIdx].Data := _readToolData.OutCmd.ToolData;         
        _toolData[_rSyncIdx].Data := _readToolData.OutCmd.ToolData;
         // set available bit
         ToolData[_rSyncIdx].Available := TRUE;
        _toolData[_rSyncIdx].Available := TRUE;
         // set timeout
         SetTimeout(PT := _rTimeout, rTimer := _rTimer);
         // inc step counter
        _rStep := 10; // -> jump to after startup           
       ELSE
         // check error ? 
         IF (_readToolData.Error)
         THEN
           ErrorID     := _readToolData.ErrorID;
           ErrorAddTxt := _readToolData.ErrorAddTxt;           
           // reset available bit
           ToolData[_rSyncIdx].Available := FALSE;
          _toolData[_rSyncIdx].Available := FALSE;
         END_IF  
       
         // timeout exceeded ? 
         IF (CheckTimeout(_rTimer) = RobotLibraryConstants.OK)
         THEN
           ErrorID     := RobotLibraryErrorIdEnum.ERR_TIMEOUT_CMD;
           ErrorAddTxt := CONCAT(_stepName, DINT_TO_STRING(_rStep));
         END_IF
       END_IF


  // ------------------------------------------
  // Write data from PLC to RC
  // ------------------------------------------
  30 : IF (( NOT _writeToolData.Busy  ) AND 
           ( NOT _writeToolData.Error ))
       THEN
         // set command parameter
        _writeToolData.ParCmd.ToolNo   := _rSyncIdx;      
        _writeToolData.ParCmd.ToolData :=  ToolData[_rSyncIdx].Data;
         // execute command
        _writeToolData.Execute := TRUE;
         // set timeout
         SetTimeout(PT := _rTimeout, rTimer := _rTimer);
         // inc step counter
        _rStep := _rStep + 1;
       ELSE
         // check error ? 
         IF (_writeToolData.Error)
         THEN
           ErrorID     := _writeToolData.ErrorID;
           ErrorAddTxt := _writeToolData.ErrorAddTxt;;
         END_IF  
       
         // timeout exceeded ? 
         IF (CheckTimeout(_rTimer) = RobotLibraryConstants.OK)
         THEN
           ErrorID     := RobotLibraryErrorIdEnum.ERR_TIMEOUT_CMD;
           ErrorAddTxt := CONCAT(_stepName, DINT_TO_STRING(_rStep));
         END_IF
       END_IF
 
  31 : IF (( NOT _writeToolData.Busy  ) AND
           ( NOT _writeToolData.Error ) AND
           (     _writeToolData.Done  ))
       THEN
         // execute command
        _writeToolData.Execute := FALSE;      
         // update internal tool data
        _toolData[_rSyncIdx] := ToolData[_rSyncIdx]; 
         // set available bit
         ToolData[_rSyncIdx].Available := TRUE; 
        _toolData[_rSyncIdx].Available := TRUE;         
         // set timeout
         SetTimeout(PT := _rTimeout, rTimer := _rTimer);
         // inc step counter
        _rStep := 10; // -> jump to after startup;           
       ELSE
         // check error ? 
         IF (_writeToolData.Error)
         THEN
           SetWarning( WarningID := RobotLibraryWarningIdEnum.WARN_TOOL_SYNC_FAILED_BY_ERROR_OF_READ_OR_WRITE_CMD, Overwrite := TRUE);    
           // reset available bit
           ToolData[_rSyncIdx].Available := FALSE;
          _toolData[_rSyncIdx].Available := FALSE;
         END_IF  
       
         // timeout exceeded ? 
         IF (CheckTimeout(_rTimer) = RobotLibraryConstants.OK)
         THEN
           ErrorID     := RobotLibraryErrorIdEnum.ERR_TIMEOUT_CMD;
           ErrorAddTxt := CONCAT(_stepName, DINT_TO_STRING(_rStep));
         END_IF
       END_IF
       
ELSE
  // invalid step
  ErrorID     := RobotLibraryErrorIdEnum.ERR_INVALID_STEP;
  ErrorAddTxt := CONCAT(_stepName , DINT_TO_STRING(_stepCmd));
END_CASE  
                
END_METHOD

METHOD PRIVATE HandleSyncWorkArea
VAR_IN_OUT
   /// Robot assignment of function
  AxesGroup : AxesGroup;
  /// Work areas stored on PLC. For more information refer to 5.5.8
  WorkAreas : ARRAY[*] OF RobotWorkArea;
END_VAR 

VAR
  /// Internal step counter name
 _stepName        : STRING;    
  /// Internal reference to step counter
 _rStep           : REFERENCE TO DINT;
  /// Internal reference to timer
 _rTimer          : REFERENCE TO TON;
  /// Internal reference to timeout
 _rTimeout        : REFERENCE TO TIME; 
  /// Internal reference to synchroniztion index
 _rSyncIdx        : REFERENCE TO USINT;
  /// internal bit for condition found
 _found           : BOOL;
  /// empty data set to reset all DataChanged bits
 _dataChangedNone : AxesGroupStateDataChanged;
  /// internal index for loops
 _idx             : DINT;
END_VAR
                  // Set internal references 
_stepName      :=   '_stepSyncWorkArea = ';
_rStep       REF=    _stepSyncWorkArea;
_rTimer      REF=   _timerSyncWorkArea;
_rTimeout    REF= _timeoutSyncWorkArea;
_rSyncIdx    REF=     _syncIdxWorkArea;

CASE _rStep
OF    
  0: // Check initialisation configured ?
     IF (( _parCfg.PLC.Parameter.SynchronizationModes.WorkAreas[SyncTime.DURING_START_UP] = SyncMode.NO_SYNCHRONIZATION ) AND
         ( _parCfg.PLC.Parameter.SynchronizationModes.WorkAreas[SyncTime. AFTER_START_UP] = SyncMode.NO_SYNCHRONIZATION ))
     THEN
       RETURN;
     END_IF
     
     // Check More Data on RC than on PLC -> Synchronization not possible
     IF (AxesGroup.State.ConfigurationData.HighestWorkAreaIndex > AxesGroup.SystemData.WorkAreasCount)
     THEN
       SetError( ErrorID := RobotLibraryErrorIdEnum.ERR_SYNC_WORKAREA_COUNT_RC_HIGHER_THAN_PLC, Overwrite := FALSE);
       RETURN;
		 END_IF
     
     // wait for initialisation done
     IF  ((     AxesGroup.State.RobotData.RCSupportedFunctions. ReadWorkArea ) AND
          (     AxesGroup.State.RobotData.RCSupportedFunctions.WriteWorkArea ) AND
          (     AxesGroup.State.Initialized                                  ) AND 
          ( NOT Error                                                        ))  
     THEN
       // Check PLC WorkAreas < RC WorkAreas and SyncWorkArea enabled ?    
       IF (( AxesGroup.State.DataEnableSync.EnableSyncWorkArea      = TRUE                              )  AND
           ( AxesGroup.Parameter.Rob.Parameter.HighestWorkAreaIndex > AxesGroup.SystemData.WorkAreasMax ))        
       THEN
         SetWarning( WarningID := RobotLibraryWarningIdEnum.WARN_WORK_AREA_ARRAY_TOO_SHORT, Overwrite := TRUE);
       END_IF

       // Create log entry
       CreateLogMessagePara1 ( Timestamp   := SystemTime,
                               MessageType := MessageType.CMD,
                               Severity    := Severity.DEBUG,
                               MessageCode := 0,
                               MessageText := 'SyncWorkArea: Start initial reading of WorkArea from RC',
                               Para1       :=  '');
       
       // init WorkArea number
      _rSyncIdx := DINT_TO_USINT(AxesGroup.SystemData.WorkAreasMin); 
       // init count of unsynchronized elements
       AxesGroup.State.SyncStatePlc.UnSyncNo.WorkArea := 0;
       // set timeout
       SetTimeout(PT := _rTimeout, rTimer := _rTimer);
       // inc step counter
      _rStep := _rStep + 1;
     END_IF     

     
     // Start read WorkArea
  1: IF (( NOT _readWorkArea.Busy  ) AND 
         ( NOT _readWorkArea.Error ) AND
         ( NOT _readWorkArea.Done  ))
     THEN
       // set command parameter
      _readWorkArea.ParCmd.WorkAreaNo := _rSyncIdx;      
       // execute command
      _readWorkArea.Execute := TRUE;
       // set timeout
       SetTimeout(PT := _rTimeout, rTimer := _rTimer);
       // inc step counter
      _rStep := _rStep + 1;
     ELSE
       // check error ? 
       IF ( _readWorkArea.Error ) 
       THEN
         SetWarning ( WarningID := RobotLibraryWarningIdEnum.WARN_WORK_AREA_SYNC_FAILED_BY_ERROR_OF_READ_OR_WRITE_CMD, Overwrite := FALSE );           
       END_IF  
       
       // timeout exceeded ? 
       IF (CheckTimeout(_rTimer) = RobotLibraryConstants.OK)
       THEN
         ErrorID     := RobotLibraryErrorIdEnum.ERR_TIMEOUT_CMD;
         ErrorAddTxt := CONCAT(_stepName, DINT_TO_STRING(_rStep));
       END_IF
     END_IF
 
     
     // Wait WorkArea read
  2: IF (( NOT _readWorkArea.Busy  ) AND
         ( NOT _readWorkArea.Error ) AND
         (     _readWorkArea.Done  ))
     THEN
       // reset execution
      _readWorkArea.Execute := FALSE;
       // set available bit
      _workAreas[_rSyncIdx].Available := TRUE; 
       WorkAreas[_rSyncIdx].Available := TRUE;      
       // Copy data
      _workAreas[_rSyncIdx].Data := _readWorkArea.OutCmd.WorkAreaData;

       // Check WorkArea data is equal ? 
       IF ( NOT IsWorkAreaEqual( Data1 := _workAreas[_rSyncIdx].Data, Data2 := WorkAreas[_rSyncIdx].Data, IgnoreTimestamp := TRUE))
       THEN
         // Reset plc in sync flag
         AxesGroup.State.SyncStatePlc.InSync.WorkArea := FALSE;
         // Set data changed flag
         AxesGroup.State.DataChanged.WorkArea[_rSyncIdx] := TRUE;
         // inc count of unsynchronised plc WorkAreas
         AxesGroup.State.SyncStatePlc.UnSyncNo.WorkArea := AxesGroup.State.SyncStatePlc.UnSyncNo.WorkArea + 1;
        
         // Create log entry
         CreateLogMessagePara1 ( Timestamp   := SystemTime,
                                 MessageType := MessageType.CMD,
                                 Severity    := Severity.DEBUG,
                                 MessageCode := 0,
                                 MessageText := 'SyncWorkArea: Detected a difference in WorkArea[{1}] between PLC and RC',
                                 Para1       :=  DINT_TO_STRING(_rSyncIdx));
        
        
         // Check synchronisation is enabled ? 
         IF ( NOT AxesGroup.State.DataEnableSync.EnableSyncWorkArea )
         THEN
           SetInfo ( InfoID := RobotLibraryInfoIdEnum.INFO_SYNC_WORK_AREA_DISABLED, Overwrite := FALSE );
				 END_IF
         
         // Check user interaction needed ?  
         IF ( AxesGroup.Parameter.PLC.Parameter.SyncUserInteraction.WorkAreas )
         THEN
           SetWarning ( WarningID := RobotLibraryWarningIdEnum.WARN_WORK_AREA_NUMBER_SYNC_ERROR, Overwrite := FALSE );                    
				 END_IF
			 END_IF
             
       // Check all WorkAreas read ? 
       IF ( _rSyncIdx < AxesGroup.State.UnifiedWorkAreaIndex )
       THEN
         // set timeout
         SetTimeout(PT := _rTimeout, rTimer := _rTimer);
         // inc WorkArea index
        _rSyncIdx := _rSyncIdx + 1;
         // dec step counter
        _rStep := _rStep - 1;
       ELSE
         // set timeout
         SetTimeout(PT := _rTimeout, rTimer := _rTimer);
         // inc step counter
        _rStep := _rStep + 1;           
       END_IF
     ELSE
       // check error ? 
       IF (_readWorkArea.Error)
       THEN
         // Set warning
         SetWarning( WarningID := RobotLibraryWarningIdEnum.WARN_WORK_AREA_SYNC_FAILED_BY_ERROR_OF_READ_OR_WRITE_CMD, Overwrite := TRUE);                    
         // reset available bit
         WorkAreas[_rSyncIdx].Available := FALSE;
        _workAreas[_rSyncIdx].Available := FALSE;
       END_IF  
       
       // timeout exceeded ? 
       IF (CheckTimeout(_rTimer) = RobotLibraryConstants.OK)
       THEN
         ErrorID     := RobotLibraryErrorIdEnum.ERR_TIMEOUT_CMD;
         ErrorAddTxt := CONCAT(_stepName, DINT_TO_STRING(_rStep));
       END_IF
     END_IF
     
     
     // Check synchronisation state ? 
  3: IF (( AxesGroup.State.SyncStatePlc.UnSyncNo.WorkArea                                             = 0                           ) OR 
         ( AxesGroup.Parameter.Plc.Parameter.SynchronizationModes.WorkAreas[SyncTime.DURING_START_UP] = SyncMode.NO_SYNCHRONIZATION ))
     THEN
       // Update bit for data in sync
       AxesGroup.State.SyncStatePlc.InSync.WorkArea := (AxesGroup.State.SyncStatePlc.UnSyncNo.WorkArea = 0);
       // set timeout
       SetTimeout(PT := _rTimeout, rTimer := _rTimer);
       // inc step counter
      _rStep := 10; // -> jump to after startup
            
       // Create log entry
       CreateLogMessagePara1 ( Timestamp   := SystemTime,
                               MessageType := MessageType.CMD,
                               Severity    := Severity.DEBUG,
                               MessageCode := 0,
                               MessageText := 'SyncWorkArea: Synchronization Startup Phase done',
                               Para1       :=  '' );      
     ELSE 
       // Check user interaction needed ? 
       IF ( NOT AxesGroup.Parameter.PLC.Parameter.SyncUserInteraction.WorkAreas )
       THEN
         CASE AxesGroup.Parameter.Plc.Parameter.SynchronizationModes.WorkAreas[SyncTime.DURING_START_UP] OF

           SyncMode.SERVER_TO_CLIENT : 

             // Overwrite PLC data with RC data
             FOR _idx := AxesGroup.SystemData.WorkAreasMin TO AxesGroup.SystemData.WorkAreasMax
             DO
               // Overwrite PLC data with RC data
               WorkAreas[_idx] := WorkAreas[_idx];            
						 END_FOR
  
             // Reset data changed flags
             AxesGroup.State.DataChanged.WorkArea := _dataChangedNone.WorkArea;
             // Reset Synchronizing flag
             AxesGroup.State.Synchronizing.WorkAreas := FALSE;
             // Set plc in sync flag
             AxesGroup.State.SyncStatePlc.InSync.WorkArea := TRUE;
             // Reset count of unsynchronised plc WorkAreas
             AxesGroup.State.SyncStatePlc.UnSyncNo.WorkArea := 0;            
             // set timeout
             SetTimeout(PT := _rTimeout, rTimer := _rTimer);
             // inc step counter
            _rStep := 10; // -> jump to after startup         

            // Create log entry
            CreateLogMessagePara3 ( Timestamp   := SystemTime,
                                    MessageType := MessageType.CMD,
                                    Severity    := Severity.DEBUG,
                                    MessageCode := 0,
                                    MessageText := 'SyncWorkArea: Synchronization of WorkAreas triggered by StartUp-Compare, SyncMode = {2}, SyncTime = {3}, SyncDirection = RC -> PLC',
                                    Para1       :=  DINT_TO_STRING(_rSyncIdx),
                                    Para2       :=  SYNC_MODE_TO_STRING(AxesGroup.Parameter.Plc.Parameter.SynchronizationModes.WorkAreas[SyncTime.DURING_START_UP]),
                                    Para3       :=  SYNC_TIME_TO_STRING(SyncTime.DURING_START_UP));
            // Create log entry
            CreateLogMessagePara1 ( Timestamp   := SystemTime,
                                    MessageType := MessageType.CMD,
                                    Severity    := Severity.DEBUG,
                                    MessageCode := 0,
                                    MessageText := 'SyncWorkArea: Applied the initial read WorkArea data from RC',
                                    Para1       :=  '' );

				   SyncMode.CLIENT_TO_SERVER : ;

             // Check conflicts to solve ? 
             FOR _rSyncIdx := 0 TO AxesGroup.State.UnifiedWorkAreaIndex
             DO
               IF ( AxesGroup.State.DataChanged.WorkArea[_rSyncIdx] )
               THEN
                _found := TRUE;
                 EXIT;
		  			   END_IF
             END_FOR
           
             IF ( _found ) 
             THEN
               // Reset plc in sync flag
               AxesGroup.State.SyncStatePlc.InSync.WorkArea := FALSE;
               // Set Synchronizing flag
               AxesGroup.State.Synchronizing.WorkAreas := TRUE;
               // set timeout
               SetTimeout(PT := _rTimeout, rTimer := _rTimer);
               // inc step counter
              _rStep := _rStep +1; // -> write PLC data to RC                  
               // Create log entry
               CreateLogMessagePara3 ( Timestamp   := SystemTime,
                                       MessageType := MessageType.CMD,
                                       Severity    := Severity.DEBUG,
                                       MessageCode := 0,
                                       MessageText := 'SyncWorkArea: Synchronization of WorkArea[{1}] triggered by StartUp-Compare, SyncMode = {2}, SyncTime = {3}, SyncDirection = PLC -> RC',
                                       Para1       :=  DINT_TO_STRING(_rSyncIdx),
                                       Para2       :=  SYNC_MODE_TO_STRING(AxesGroup.Parameter.Plc.Parameter.SynchronizationModes.WorkAreas[SyncTime.DURING_START_UP]),
                                       Para3       :=  SYNC_TIME_TO_STRING(SyncTime.DURING_START_UP));
             ELSE
               // Reset data changed flags
               AxesGroup.State.DataChanged.WorkArea := _dataChangedNone.WorkArea;
               // Reset Synchronizing flag
               AxesGroup.State.Synchronizing.WorkAreas := FALSE;
               // Set plc in sync flag
               AxesGroup.State.SyncStatePlc.InSync.WorkArea := TRUE;
               // Reset count of unsynchronised WorkAreas
               AxesGroup.State.SyncStatePlc.UnSyncNo.WorkArea := 0;
               // set timeout
               SetTimeout(PT := _rTimeout, rTimer := _rTimer);
               // inc step counter
              _rStep := 10; // -> jump to after startup                  
				     END_IF
         ELSE
           // invalid sync mode for startup
           SetError( ErrorID := RobotLibraryErrorIdEnum.ERR_SYNC_MODE_INVALID, Overwrite := TRUE );
 	       END_CASE
       END_IF
     END_IF  

     
     // Start write WorkArea data  
  4: IF (( NOT _writeWorkArea.Busy  ) AND 
         ( NOT _writeWorkArea.Error ))
     THEN
       // set command parameter
      _writeWorkArea.ParCmd.WorkAreaNo   := _rSyncIdx;      
      _writeWorkArea.ParCmd.WorkAreaData :=  WorkAreas[_rSyncIdx].Data;
       // execute command
      _writeWorkArea.Execute := TRUE;
       // set timeout
       SetTimeout(PT := _rTimeout, rTimer := _rTimer);
       // inc step counter
      _rStep := _rStep + 1;
     ELSE
       // check error ? 
       IF (_writeWorkArea.Error)
       THEN
         ErrorID     := _writeWorkArea.ErrorID;
         ErrorAddTxt := _writeWorkArea.ErrorAddTxt;;
       END_IF  
       
       // timeout exceeded ? 
       IF (CheckTimeout(_rTimer) = RobotLibraryConstants.OK)
       THEN
         ErrorID     := RobotLibraryErrorIdEnum.ERR_TIMEOUT_CMD;
         ErrorAddTxt := CONCAT(_stepName, DINT_TO_STRING(_rStep));
       END_IF
     END_IF
 
     
     // Wait WorkArea data written ?   
  5: IF (( NOT _writeWorkArea.Busy  ) AND
         ( NOT _writeWorkArea.Error ) AND
         (     _writeWorkArea.Done  ))
     THEN
       // execute command
      _writeWorkArea.Execute := FALSE;
       // apply WorkArea data to internal WorkArea data
      _workAreas[_rSyncIdx] := WorkAreas[_rSyncIdx];
       // reset data changed bit 
       AxesGroup.State.DataChanged.WorkArea[_rSyncIdx] := FALSE;
       // dec count of unsynchronised WorkAreas
       AxesGroup.State.SyncStatePlc.UnSyncNo.WorkArea := AxesGroup.State.SyncStatePlc.UnSyncNo.WorkArea - 1;
       // set timeout        
       SetTimeout(PT := _rTimeout, rTimer := _rTimer);
       // dec step counter
      _rStep := _rStep - 2; 
     ELSE
       // check error ? 
       IF (_writeWorkArea.Error)
       THEN
         SetWarning( WarningID := RobotLibraryWarningIdEnum.WARN_WORK_AREA_SYNC_FAILED_BY_ERROR_OF_READ_OR_WRITE_CMD, Overwrite := TRUE);           
       END_IF  
       
       // timeout exceeded ? 
       IF (CheckTimeout(_rTimer) = RobotLibraryConstants.OK)
       THEN
         ErrorID     := RobotLibraryErrorIdEnum.ERR_TIMEOUT_CMD;
         ErrorAddTxt := CONCAT(_stepName, DINT_TO_STRING(_rStep));
       END_IF
     END_IF

     
  // --------------------------------------------
  // SyncMode after startup : 
  // --------------------------------------------
         
  10 : // check synchronisation active ? 
       IF ( AxesGroup.Parameter.Plc.Parameter.SynchronizationModes.WorkAreas[SyncTime.AFTER_START_UP] = SyncMode.NO_SYNCHRONIZATION)
       THEN
         RETURN;
       END_IF
       
       // reset count of unsynchronised WorkAreas
       AxesGroup.State.SyncStatePlc.UnSyncNo.WorkArea := 0;

       // Check all WorkArea datas
       FOR _rSyncIdx := 0 TO AxesGroup.State.UnifiedWorkAreaIndex
       DO
         // compare WorkArea data
         AxesGroup.State.DataChanged.WorkArea[_rSyncIdx] := NOT IsWorkAreaEqual( Data1 := WorkAreas[_rSyncIdx].Data, Data2 := _workAreas[_rSyncIdx].Data, IgnoreTimestamp := FALSE);

         // Check WorkArea data changed ? 
         IF (AxesGroup.State.DataChanged.WorkArea[_rSyncIdx])
         THEN
           // inc count of unsynchronised plc WorkAreas
           AxesGroup.State.SyncStatePlc.UnSyncNo.WorkArea := AxesGroup.State.SyncStatePlc.UnSyncNo.WorkArea + 1;
           // Create log entry
           CreateLogMessagePara2 ( Timestamp   := SystemTime,
                                   MessageType := MessageType.CMD,
                                   Severity    := Severity.DEBUG,
                                   MessageCode := 0,
                                   MessageText := 'SyncWorkArea: Detected a local change of WorkArea[{1}] on PLC, SyncTime = {2}',
                                   Para1       :=  DINT_TO_STRING(_rSyncIdx),    
                                   Para2       :=  SYNC_TIME_TO_STRING(SyncTime.AFTER_START_UP));       
				 END_IF

         // Update plc in sync flag
         AxesGroup.State.SyncStatePlc.InSync.WorkArea := (AxesGroup.State.SyncStatePlc.UnSyncNo.WorkArea = 0); 
	     END_FOR

       // Check synchronization is needed ? 
       IF ( NOT AxesGroup.State.SyncStatePlc.InSync.WorkArea ) XOR  
          ( NOT AxesGroup.State.SyncStateRc .InSync.WorkArea )
       THEN
         CASE AxesGroup.Parameter.Plc.Parameter.SynchronizationModes.WorkAreas[SyncTime.AFTER_START_UP] 
         OF         
           // NO_SYNCHRONIZATION
           SyncMode.NO_SYNCHRONIZATION : ; // no further action 
           
           // CLIENT_TO_SERVER
           SyncMode.CLIENT_TO_SERVER :
             // set timeout
             SetTimeout(PT := _rTimeout, rTimer := _rTimer);
             // inc step counter
            _rStep := 11;
  
           // SERVER_TO_CLIENT
           SyncMode.SERVER_TO_CLIENT :
             // set timeout
             SetTimeout(PT := _rTimeout, rTimer := _rTimer);
             // inc step counter
            _rStep := 12;
  
           // AUTOMATIC
           SyncMode.AUTOMATIC : 
             // set timeout
             SetTimeout(PT := _rTimeout, rTimer := _rTimer);
             // inc step counter
            _rStep := 13;
         END_CASE
       ELSE
         // datas changeḍ on both sides ? -> Warning 
         IF (( NOT AxesGroup.State.SyncStatePlc.InSync.WorkArea ) AND  
             ( NOT AxesGroup.State.SyncStateRc .InSync.WorkArea ))
         THEN
           SetWarning( WarningID := RobotLibraryWarningIdEnum.WARN_WORK_AREA_SYNC_BOTH_SIDES_CHANGED, Overwrite := TRUE);
         END_IF
       END_IF


  // ------------------------------------------
  // SyncMode : CLIENT_TO_SERVER 
  // ------------------------------------------  
  11 : // Conflict triggerd by PLC ?  
       IF ( NOT AxesGroup.State.SyncStatePlc.InSync.WorkArea )
       THEN
         // search for changed index  
         FOR _rSyncIdx := 0 TO AxesGroup.State.UnifiedWorkAreaIndex
         DO
           IF ( AxesGroup.State.DataChanged.WorkArea[_rSyncIdx] )
           THEN
             // set timeout
             SetTimeout(PT := _rTimeout, rTimer := _rTimer);
             // inc step counter
            _rStep := 30; // -> write PLC data to RC                  
             EXIT;             
					 END_IF
         END_FOR
         
         // Create log entry
         CreateLogMessagePara3 ( Timestamp   := SystemTime,
                                 MessageType := MessageType.CMD,
                                 Severity    := Severity.DEBUG,
                                 MessageCode := 0,
                                 MessageText := 'SyncWorkArea: Synchronization of WorkArea[{1}] triggered by PLC, SyncMode = {2}, SyncTime = {3}, SyncDirection = PLC -> RC',
                                 Para1       :=  DINT_TO_STRING(_rSyncIdx),
                                 Para2       :=  SYNC_MODE_TO_STRING(AxesGroup.Parameter.Plc.Parameter.SynchronizationModes.WorkAreas[SyncTime.AFTER_START_UP]),
                                 Para3       :=  SYNC_TIME_TO_STRING(SyncTime.AFTER_START_UP));
                                 RETURN;
       END_IF
   
       // Conflict triggered by RC ?
       IF ( NOT AxesGroup.State.SyncStateRc.InSync.WorkArea )
       THEN
         // get changed index 
        _rSyncIdx :=  LIMIT(0, AxesGroup.State.SyncStateRc.UnSyncNo.WorkArea, AxesGroup.State.UnifiedWorkAreaIndex);
         // set timeout
         SetTimeout(PT := _rTimeout, rTimer := _rTimer);
         // inc step counter
        _rStep := 30; // -> write PLC data to RC

         // Create log entry
         CreateLogMessagePara3 ( Timestamp   := SystemTime,
                                 MessageType := MessageType.CMD,
                                 Severity    := Severity.DEBUG,
                                 MessageCode := 0,
                                 MessageText := 'SyncWorkArea: Synchronization of WorkArea[{1}] triggered by RC, SyncMode = {2}, SyncTime = {3}, SyncDirection = PLC -> RC',
                                 Para1       :=  DINT_TO_STRING(_rSyncIdx),
                                 Para2       :=  SYNC_MODE_TO_STRING(AxesGroup.Parameter.Plc.Parameter.SynchronizationModes.WorkAreas[SyncTime.AFTER_START_UP]),
                                 Para3       :=  SYNC_TIME_TO_STRING(SyncTime.AFTER_START_UP));
                                 RETURN;
			 END_IF
       
       // set timeout
       SetTimeout(PT := _rTimeout, rTimer := _rTimer);
       // jump back
      _rStep := 10;

       
  // ------------------------------------------
  // SyncMode : SERVER_TO_CLIENT 
  // ------------------------------------------
  12 : // Conflict triggerd by PLC ?  
       IF ( NOT AxesGroup.State.SyncStatePlc.InSync.WorkArea )
       THEN
         // search for changed index  
         FOR _rSyncIdx := 0 TO AxesGroup.State.UnifiedWorkAreaIndex
         DO
           IF ( AxesGroup.State.DataChanged.WorkArea[_rSyncIdx] )
           THEN
             // set timeout
             SetTimeout(PT := _rTimeout, rTimer := _rTimer);
             // inc step counter
            _rStep := 20; // -> read RC data and write it to PLC                  
             EXIT;
					 END_IF
         END_FOR

         // Create log entry
         CreateLogMessagePara3 ( Timestamp   := SystemTime,
                                 MessageType := MessageType.CMD,
                                 Severity    := Severity.DEBUG,
                                 MessageCode := 0,
                                 MessageText := 'SyncWorkArea: Synchronization of WorkArea[{1}] triggered by PLC, SyncMode = {2}, SyncTime = {3}, SyncDirection = RC -> PLC',
                                 Para1       :=  DINT_TO_STRING(_rSyncIdx),
                                 Para2       :=  SYNC_MODE_TO_STRING(AxesGroup.Parameter.Plc.Parameter.SynchronizationModes.WorkAreas[SyncTime.AFTER_START_UP]),
                                 Para3       :=  SYNC_TIME_TO_STRING(SyncTime.AFTER_START_UP));
                                 RETURN;
       END_IF
   
       // Conflict triggered by RC ?
       IF ( NOT AxesGroup.State.SyncStateRc.InSync.WorkArea )
       THEN
         // get changed index 
        _rSyncIdx := LIMIT(0, AxesGroup.State.SyncStateRc.UnSyncNo.WorkArea, AxesGroup.State.UnifiedWorkAreaIndex);
         // set timeout
         SetTimeout(PT := _rTimeout, rTimer := _rTimer);
         // inc step counter
        _rStep := 20; // -> read RC data and write it to PLC

         // Create log entry
         CreateLogMessagePara3 ( Timestamp   := SystemTime,
                                 MessageType := MessageType.CMD,
                                 Severity    := Severity.DEBUG,
                                 MessageCode := 0,
                                 MessageText := 'SyncWorkArea: Synchronization of WorkArea[{1}] triggered by RC, SyncMode = {2}, SyncTime = {3}, SyncDirection = RC -> PLC',
                                 Para1       :=  DINT_TO_STRING(_rSyncIdx),
                                 Para2       :=  SYNC_MODE_TO_STRING(AxesGroup.Parameter.Plc.Parameter.SynchronizationModes.WorkAreas[SyncTime.AFTER_START_UP]),
                                 Para3       :=  SYNC_TIME_TO_STRING(SyncTime.AFTER_START_UP));
                                 RETURN;
			 END_IF
       
       // set timeout
       SetTimeout(PT := _rTimeout, rTimer := _rTimer);
       // jump back
      _rStep := 10;
  

  // ------------------------------------------
  // SyncMode : AUTOMATIC 
  // ------------------------------------------
  13 : // Conflict triggerd by PLC ?  
       IF ( NOT AxesGroup.State.SyncStatePlc.InSync.WorkArea )
       THEN
         // search for changed index  
         FOR _rSyncIdx := 0 TO AxesGroup.State.UnifiedWorkAreaIndex
         DO
           IF ( AxesGroup.State.DataChanged.WorkArea[_rSyncIdx] )
           THEN
             // set timeout
             SetTimeout(PT := _rTimeout, rTimer := _rTimer);
             // inc step counter
            _rStep := 30; // -> write PLC data to RC                  
             EXIT;
					 END_IF
         END_FOR
         
         // Create log entry
         CreateLogMessagePara3 ( Timestamp   := SystemTime,
                                 MessageType := MessageType.CMD,
                                 Severity    := Severity.DEBUG,
                                 MessageCode := 0,
                                 MessageText := 'SyncWorkArea: Synchronization of WorkArea[{1}] triggered by PLC, SyncMode = {2}, SyncTime = {3}, SyncDirection = PLC -> RC',
                                 Para1       :=  DINT_TO_STRING(_rSyncIdx),
                                 Para2       :=  SYNC_MODE_TO_STRING(AxesGroup.Parameter.Plc.Parameter.SynchronizationModes.WorkAreas[SyncTime.AFTER_START_UP]),
                                 Para3       :=  SYNC_TIME_TO_STRING(SyncTime.AFTER_START_UP));
                                 RETURN;
       END_IF
   
       // Conflict triggered by RC ?
       IF ( NOT AxesGroup.State.SyncStateRc.InSync.WorkArea )
       THEN
         // get changed index 
        _rSyncIdx := LIMIT(0, AxesGroup.State.SyncStateRc.UnSyncNo.WorkArea, AxesGroup.State.UnifiedWorkAreaIndex);
         // set timeout
         SetTimeout(PT := _rTimeout, rTimer := _rTimer);
         // inc step counter
        _rStep := 20; // -> read RC data an write it to PLC

         // Create log entry
         CreateLogMessagePara3 ( Timestamp   := SystemTime,
                                 MessageType := MessageType.CMD,
                                 Severity    := Severity.DEBUG,
                                 MessageCode := 0,
                                 MessageText := 'SyncWorkArea: Synchronization of WorkArea[{1}] triggered by RC, SyncMode = {2}, SyncTime = {3}, SyncDirection = RC -> PLC',
                                 Para1       :=  DINT_TO_STRING(_rSyncIdx),
                                 Para2       :=  SYNC_MODE_TO_STRING(AxesGroup.Parameter.Plc.Parameter.SynchronizationModes.WorkAreas[SyncTime.AFTER_START_UP]),
                                 Para3       :=  SYNC_TIME_TO_STRING(SyncTime.AFTER_START_UP));
                                 RETURN;
			 END_IF
       
       // set timeout
       SetTimeout(PT := _rTimeout, rTimer := _rTimer);
       // jump back
      //_rStep := 10;


  // ------------------------------------------
  // Read Data from RC and write it to PLC
  // ------------------------------------------
  20 : IF (( NOT _readWorkArea.Busy  ) AND 
           ( NOT _readWorkArea.Error ))
       THEN
         // set command parameter
        _readWorkArea.ParCmd.WorkAreaNo := _rSyncIdx;      
         // execute command
        _readWorkArea.Execute := TRUE;
         // set timeout
         SetTimeout(PT := _rTimeout, rTimer := _rTimer);
         // inc step counter
        _rStep := _rStep + 1;
       ELSE
         // check error ? 
         IF (_readWorkArea.Error)
         THEN
           ErrorID     := _readWorkArea.ErrorID;
           ErrorAddTxt := _readWorkArea.ErrorAddTxt;
         END_IF  
       
         // timeout exceeded ? 
         IF (CheckTimeout(_rTimer) = RobotLibraryConstants.OK)
         THEN
           ErrorID     := RobotLibraryErrorIdEnum.ERR_TIMEOUT_CMD;
           ErrorAddTxt := CONCAT(_stepName, DINT_TO_STRING(_rStep));
         END_IF
       END_IF
 
  21 : IF (( NOT _readWorkArea.Busy  ) AND
           ( NOT _readWorkArea.Error ) AND
           (     _readWorkArea.Done  ))
       THEN
         // reset execution
        _readWorkArea.Execute := FALSE;
         // update internal WorkArea data
         WorkAreas[_rSyncIdx].Data := _readWorkArea.OutCmd.WorkAreaData;         
        _workAreas[_rSyncIdx].Data := _readWorkArea.OutCmd.WorkAreaData;
         // set available bit
         WorkAreas[_rSyncIdx].Available := TRUE;
        _workAreas[_rSyncIdx].Available := TRUE;
         // set timeout
         SetTimeout(PT := _rTimeout, rTimer := _rTimer);
         // inc step counter
        _rStep := 10; // -> jump to after startup           
       ELSE
         // check error ? 
         IF (_readWorkArea.Error)
         THEN
           ErrorID     := _readWorkArea.ErrorID;
           ErrorAddTxt := _readWorkArea.ErrorAddTxt;           
           // reset available bit
           WorkAreas[_rSyncIdx].Available := FALSE;
          _workAreas[_rSyncIdx].Available := FALSE;
         END_IF  
       
         // timeout exceeded ? 
         IF (CheckTimeout(_rTimer) = RobotLibraryConstants.OK)
         THEN
           ErrorID     := RobotLibraryErrorIdEnum.ERR_TIMEOUT_CMD;
           ErrorAddTxt := CONCAT(_stepName, DINT_TO_STRING(_rStep));
         END_IF
       END_IF


  // ------------------------------------------
  // Write data from PLC to RC
  // ------------------------------------------
  30 : IF (( NOT _writeWorkArea.Busy  ) AND 
           ( NOT _writeWorkArea.Error ))
       THEN
         // set command parameter
        _writeWorkArea.ParCmd.WorkAreaNo   := _rSyncIdx;      
        _writeWorkArea.ParCmd.WorkAreaData :=  WorkAreas[_rSyncIdx].Data;
         // execute command
        _writeWorkArea.Execute := TRUE;
         // set timeout
         SetTimeout(PT := _rTimeout, rTimer := _rTimer);
         // inc step counter
        _rStep := _rStep + 1;
       ELSE
         // check error ? 
         IF (_writeWorkArea.Error)
         THEN
           ErrorID     := _writeWorkArea.ErrorID;
           ErrorAddTxt := _writeWorkArea.ErrorAddTxt;;
         END_IF  
       
         // timeout exceeded ? 
         IF (CheckTimeout(_rTimer) = RobotLibraryConstants.OK)
         THEN
           ErrorID     := RobotLibraryErrorIdEnum.ERR_TIMEOUT_CMD;
           ErrorAddTxt := CONCAT(_stepName, DINT_TO_STRING(_rStep));
         END_IF
       END_IF
 
  31 : IF (( NOT _writeWorkArea.Busy  ) AND
           ( NOT _writeWorkArea.Error ) AND
           (     _writeWorkArea.Done  ))
       THEN
         // execute command
        _writeWorkArea.Execute := FALSE;      
         // update internal WorkArea data
        _workAreas[_rSyncIdx] := WorkAreas[_rSyncIdx]; 
         // set available bit
         WorkAreas[_rSyncIdx].Available := TRUE; 
        _workAreas[_rSyncIdx].Available := TRUE;         
         // set timeout
         SetTimeout(PT := _rTimeout, rTimer := _rTimer);
         // inc step counter
        _rStep := 10; // -> jump to after startup;           
       ELSE
         // check error ? 
         IF (_writeWorkArea.Error)
         THEN
           SetWarning( WarningID := RobotLibraryWarningIdEnum.WARN_WORK_AREA_SYNC_FAILED_BY_ERROR_OF_READ_OR_WRITE_CMD, Overwrite :=  TRUE);    
           // reset available bit
           WorkAreas[_rSyncIdx].Available := FALSE;
          _workAreas[_rSyncIdx].Available := FALSE;
         END_IF  
       
         // timeout exceeded ? 
         IF (CheckTimeout(_rTimer) = RobotLibraryConstants.OK)
         THEN
           ErrorID     := RobotLibraryErrorIdEnum.ERR_TIMEOUT_CMD;
           ErrorAddTxt := CONCAT(_stepName, DINT_TO_STRING(_rStep));
         END_IF
       END_IF
       
ELSE
  // invalid step
  ErrorID     := RobotLibraryErrorIdEnum.ERR_INVALID_STEP;
  ErrorAddTxt := CONCAT(_stepName , DINT_TO_STRING(_stepCmd));
END_CASE  
                
END_METHOD

METHOD PRIVATE HandleTelegramStateCtrl
VAR_INPUT
END_VAR
                  // Telegram Control
// ----------------
IF ( _lastTelegramControl <> GetHalfeByteLo(Telegram.PlcToRob.Header.AxesGroupID_Control))
THEN
  // Create log entry
  CreateLogMessagePara2 ( Timestamp   := SystemTime,
                          MessageType := MessageType.CMD,
                          Severity    := Severity.INFO,
                          MessageCode := 0,
                          MessageText := 'SRCI Interface control changed from {1} to {2}',
                          Para1       := TELEGRAM_CONTROL_TO_STRING(_lastTelegramControl),
                          Para2       := TELEGRAM_CONTROL_TO_STRING(GetHalfeByteLo(Telegram.PlcToRob.Header.AxesGroupID_Control)));

  _lastTelegramControl := GetHalfeByteLo(Telegram.PlcToRob.Header.AxesGroupID_Control);
END_IF


// Telegram State
// ----------------
IF ( _lastTelegramState <> Telegram.RobToPlc.Header.TelegramState)
THEN
  // Create log entry
  CreateLogMessagePara2 ( Timestamp   := SystemTime,
                          MessageType := MessageType.CMD,
                          Severity    := Severity.INFO,
                          MessageCode := 0,
                          MessageText := 'SRCI Interface state changed from {1} to {2}',
                          Para1       := TELEGRAM_STATE_TO_STRING(_lastTelegramState),
                          Para2       := TELEGRAM_STATE_TO_STRING(Telegram.RobToPlc.Header.TelegramState));


  // Check Interface changed after being initialized ?  
  IF ((  Enable                                                                          ) AND
      ( _lastTelegramState                      = TelegramState.INITIALIZED              ) AND  
     ((  Telegram.RobToPlc.Header.TelegramState = TelegramState.READY_FOR_INITIALIZATION ) OR
      (  Telegram.RobToPlc.Header.TelegramState = TelegramState.READY_TO_RESUME          )))
  THEN
    {warning 'ToDo'}
    //SetError( ErrorID := RobotLibraryErrorIdEnum.ERR_INTERFACE_WAS_RESET_AFTER_INIT_0x80A7  , Overwrite := TRUE );
    ;
	END_IF

  // apply new telegram state
 _lastTelegramState := Telegram.RobToPlc.Header.TelegramState;
END_IF
                
END_METHOD

METHOD HandleUserData
VAR_IN_OUT
   /// Robot assignment of function
  AxesGroup    : AxesGroup;
  ///  User data stored on the PLC according to Table 6-10
  UserData     : UserData;
END_VAR
                  // Common
UserData.LogLevel                          := LogLevel;

UserData.PLCManufacturedID                 := _parCfg.Plc.Parameter.ManufacturedID;
UserData.PLCOrderID                        := _parCfg.Plc.Parameter.OrderID;
UserData.PLCSerialNumber                   := _parCfg.Plc.Parameter.SerialNumber;
UserData.PLCFirmwareVersion                := _parCfg.Plc.Parameter.FirmwareVersion;
UserData.PLCInterfaceVersion               := _parCfg.Plc.Parameter.InterfaceVersion;
UserData.PLCLibraryVersion                 :=  RobotLibraryConstants.PLCLibraryVersion;
                                           
// Communication                           
UserData.LifeSignTimeOut                   := _parCfg.Com.LifeSignTimeOut;
                                           
// Plc Parameter                           
UserData.SynchronizationModes              := _parCfg.Plc.Parameter.SynchronizationModes;
UserData.EnableSync                        :=  SyncModesToDataEnableSync(Value := _parCfg.Plc.Parameter.SynchronizationModes);
                                           
